KUKA KRL program: f1_Kuka_APT231T02S31.SRC

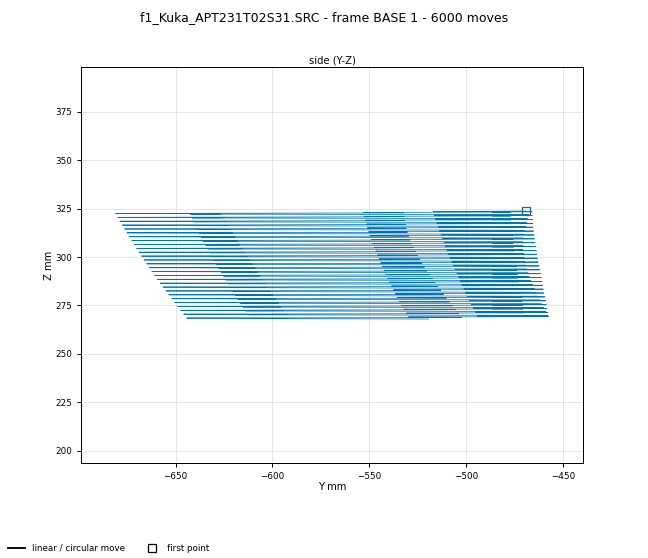
[picture p0: tool path of f1_Kuka_APT231T02S31.SRC in frame BASE 1, 6000 of 6001 moves have a stored position in this frame; points joined in program order, loops and branches not executed]
&ACCESS RVP
&REL 2
&PARAM TEMPLATE = C:\KRC\Roboter\Template\vorgabe
&PARAM EDITMASK = *
DEF f1_Kuka_APT231T02S31()


;FOLD INI;%{PE}%V3.2.0,%MKUKATPBASIS,%CINIT,%VCOMMON,%P
  ;FOLD BAS INI;%{E}%V3.2.0,%MKUKATPBASIS,%CINIT,%VINIT,%P
    GLOBAL INTERRUPT DECL 3 WHEN $STOPMESS==TRUE DO IR_STOPM ( )
    INTERRUPT ON 3
    BAS (#INITMOV,0 )
  ;ENDFOLD (BAS INI)
  ;FOLD USER INI;%{E}%V3.2.0,%MKUKATPUSER,%CINIT,%VINIT,%P
    ;Make your modifications here
  ;ENDFOLD (USER INI)
;ENDFOLD (INI)


;*** Make Null PTP Move
  PTP $pos_act

;*** Auto Load The Correct TOOL Data
  $tool=tool_data[2]

;*** Auto Load The Correct BASE Data
  $base=base_data[1]

  $ADVANCE = 5

;*** Restate Last Velocity
MMPM(30000.0)
SetRPM(8000)
LIN {X 0.027,Y -469.102,Z 323.706,A 0.000,B 0.000,C 90.000,E1 163.015} C_DIS
LIN {X -0.054,Y -471.891,Z 323.687,A 0.000,B 0.000,C 90.000,E1 159.571} C_DIS
LIN {X 0.052,Y -475.505,Z 323.669,A 0.000,B 0.000,C 90.000,E1 156.433} C_DIS
LIN {X 0.015,Y -479.747,Z 323.654,A 0.000,B 0.000,C 90.000,E1 153.640} C_DIS
LIN {X -0.289,Y -483.697,Z 323.642,A 0.000,B 0.000,C 90.000,E1 151.513} C_DIS
LIN {X -0.138,Y -490.881,Z 323.623,A 0.000,B 0.000,C 90.000,E1 148.122} C_DIS
LIN {X -0.106,Y -495.482,Z 323.613,A 0.000,B 0.000,C 90.000,E1 146.294} C_DIS
LIN {X -0.238,Y -500.846,Z 323.601,A 0.000,B 0.000,C 90.000,E1 144.196} C_DIS
LIN {X -0.122,Y -504.629,Z 323.593,A 0.000,B 0.000,C 90.000,E1 142.683} C_DIS
LIN {X 0.166,Y -507.447,Z 323.586,A 0.000,B 0.000,C 90.000,E1 141.457} C_DIS
LIN {X -0.132,Y -509.344,Z 323.581,A 0.000,B 0.000,C 90.000,E1 140.598} C_DIS
LIN {X 0.150,Y -511.693,Z 323.574,A 0.000,B 0.000,C 90.000,E1 139.380} C_DIS
LIN {X -0.165,Y -513.302,Z 323.570,A 0.000,B 0.000,C 90.000,E1 138.528} C_DIS
LIN {X 0.005,Y -514.265,Z 323.566,A 0.000,B 0.000,C 90.000,E1 137.919} C_DIS
LIN {X 0.095,Y -515.410,Z 323.561,A 0.000,B 0.000,C 90.000,E1 137.025} C_DIS
LIN {X 0.170,Y -516.215,Z 323.556,A 0.000,B 0.000,C 90.000,E1 136.134} C_DIS
LIN {X -0.015,Y -516.616,Z 323.553,A 0.000,B 0.000,C 90.000,E1 135.567} C_DIS
LIN {X -0.015,Y -516.959,Z 323.547,A 0.000,B 0.000,C 90.000,E1 134.393} C_DIS
LIN {X 0.093,Y -516.892,Z 323.542,A 0.000,B 0.000,C 90.000,E1 133.500} C_DIS
LIN {X 0.111,Y -516.371,Z 323.535,A 0.000,B 0.000,C 90.000,E1 132.324} C_DIS
LIN {X -0.152,Y -515.651,Z 323.530,A 0.000,B 0.000,C 90.000,E1 131.472} C_DIS
LIN {X -0.166,Y -514.311,Z 323.524,A 0.000,B 0.000,C 90.000,E1 130.297} C_DIS
LIN {X -0.225,Y -512.354,Z 323.516,A 0.000,B 0.000,C 90.000,E1 128.830} C_DIS
LIN {X 0.087,Y -510.241,Z 323.507,A 0.000,B 0.000,C 90.000,E1 127.317} C_DIS
LIN {X 0.041,Y -508.579,Z 323.501,A 0.000,B 0.000,C 90.000,E1 126.137} C_DIS
LIN {X 0.169,Y -507.164,Z 323.496,A 0.000,B 0.000,C 90.000,E1 125.231} C_DIS
LIN {X -0.211,Y -504.512,Z 323.488,A 0.000,B 0.000,C 90.000,E1 123.785} C_DIS
LIN {X 0.180,Y -502.175,Z 323.481,A 0.000,B 0.000,C 90.000,E1 122.546} C_DIS
LIN {X 0.128,Y -499.142,Z 323.473,A 0.000,B 0.000,C 90.000,E1 121.052} C_DIS
LIN {X 0.190,Y -496.035,Z 323.464,A 0.000,B 0.000,C 90.000,E1 119.539} C_DIS
LIN {X 0.194,Y -492.872,Z 323.456,A 0.000,B 0.000,C 90.000,E1 118.025} C_DIS
LIN {X -0.096,Y -489.685,Z 323.447,A 0.000,B 0.000,C 90.000,E1 116.539} C_DIS
LIN {X -0.219,Y -486.506,Z 323.439,A 0.000,B 0.000,C 90.000,E1 115.027} C_DIS
LIN {X 0.048,Y -483.203,Z 323.430,A 0.000,B 0.000,C 90.000,E1 113.462} C_DIS
LIN {X 0.246,Y -479.874,Z 323.422,A 0.000,B 0.000,C 90.000,E1 111.897} C_DIS
LIN {X 0.024,Y -476.568,Z 323.413,A 0.000,B 0.000,C 90.000,E1 110.375} C_DIS
LIN {X -0.039,Y -474.512,Z 323.408,A 0.000,B 0.000,C 90.000,E1 109.450} C_DIS
LIN {X -0.150,Y -469.589,Z 323.396,A 0.000,B 0.000,C 90.000,E1 107.275} C_DIS
LIN {X -0.199,Y -466.672,Z 323.389,A 0.000,B 0.000,C 90.000,E1 106.024} C_DIS
LIN {X 0.061,Y -465.888,Z 323.387,A 0.000,B 0.000,C 90.000,E1 105.662} C_DIS
LIN {X 0.021,Y -465.881,Z 323.387,A 0.000,B 0.000,C 90.000,E1 105.662} C_DIS
LIN {X -0.090,Y -467.389,Z 323.384,A 0.000,B 0.000,C 90.000,E1 105.064} C_DIS
LIN {X 0.166,Y -468.029,Z 323.382,A 0.000,B 0.000,C 90.000,E1 104.717} C_DIS
LIN {X 0.143,Y -476.239,Z 323.356,A 0.000,B 0.000,C 90.000,E1 100.018} C_DIS
LIN {X -0.072,Y -482.133,Z 323.330,A 0.000,B 0.000,C 90.000,E1 95.391} C_DIS
LIN {X 0.164,Y -485.530,Z 323.304,A 0.000,B 0.000,C 90.000,E1 90.745} C_DIS
LIN {X 0.196,Y -486.380,Z 323.280,A 0.000,B 0.000,C 90.000,E1 86.445} C_DIS
LIN {X 0.020,Y -486.349,Z 323.279,A 0.000,B 0.000,C 90.000,E1 86.159} C_DIS
LIN {X 0.099,Y -484.663,Z 323.253,A 0.000,B 0.000,C 90.000,E1 81.546} C_DIS
LIN {X -0.011,Y -480.582,Z 323.227,A 0.000,B 0.000,C 90.000,E1 76.937} C_DIS
LIN {X 0.168,Y -479.655,Z 323.224,A 0.000,B 0.000,C 90.000,E1 76.297} C_DIS
LIN {X 0.002,Y -477.055,Z 323.214,A 0.000,B 0.000,C 90.000,E1 74.574} C_DIS
LIN {X -0.038,Y -477.056,Z 323.214,A 0.000,B 0.000,C 90.000,E1 74.574} C_DIS
LIN {X -0.110,Y -479.157,Z 323.210,A 0.000,B 0.000,C 90.000,E1 73.850} C_DIS
LIN {X 0.001,Y -482.530,Z 323.203,A 0.000,B 0.000,C 90.000,E1 72.598} C_DIS
LIN {X 0.163,Y -486.664,Z 323.195,A 0.000,B 0.000,C 90.000,E1 71.040} C_DIS
LIN {X 0.125,Y -491.697,Z 323.185,A 0.000,B 0.000,C 90.000,E1 69.209} C_DIS
LIN {X -0.023,Y -497.656,Z 323.173,A 0.000,B 0.000,C 90.000,E1 67.102} C_DIS
LIN {X -0.170,Y -501.972,Z 323.164,A 0.000,B 0.000,C 90.000,E1 65.613} C_DIS
LIN {X -0.102,Y -507.999,Z 323.153,A 0.000,B 0.000,C 90.000,E1 63.512} C_DIS
LIN {X -0.093,Y -514.007,Z 323.141,A 0.000,B 0.000,C 90.000,E1 61.435} C_DIS
LIN {X 0.030,Y -518.258,Z 323.133,A 0.000,B 0.000,C 90.000,E1 59.950} C_DIS
LIN {X -0.026,Y -523.352,Z 323.123,A 0.000,B 0.000,C 90.000,E1 58.201} C_DIS
LIN {X 0.318,Y -528.367,Z 323.114,A 0.000,B 0.000,C 90.000,E1 56.421} C_DIS
LIN {X -0.074,Y -531.598,Z 323.107,A 0.000,B 0.000,C 90.000,E1 55.308} C_DIS
LIN {X 0.006,Y -535.465,Z 323.099,A 0.000,B 0.000,C 90.000,E1 53.863} C_DIS
LIN {X 0.012,Y -537.610,Z 323.095,A 0.000,B 0.000,C 90.000,E1 53.004} C_DIS
LIN {X 0.054,Y -540.270,Z 323.088,A 0.000,B 0.000,C 90.000,E1 51.859} C_DIS
LIN {X 0.024,Y -542.118,Z 323.083,A 0.000,B 0.000,C 90.000,E1 51.009} C_DIS
LIN {X -0.292,Y -544.439,Z 323.077,A 0.000,B 0.000,C 90.000,E1 49.908} C_DIS
LIN {X -0.227,Y -546.470,Z 323.071,A 0.000,B 0.000,C 90.000,E1 48.771} C_DIS
LIN {X -0.170,Y -547.848,Z 323.066,A 0.000,B 0.000,C 90.000,E1 47.919} C_DIS
LIN {X -0.062,Y -549.476,Z 323.060,A 0.000,B 0.000,C 90.000,E1 46.782} C_DIS
LIN {X -0.375,Y -550.552,Z 323.055,A 0.000,B 0.000,C 90.000,E1 45.972} C_DIS
LIN {X 0.106,Y -551.383,Z 323.051,A 0.000,B 0.000,C 90.000,E1 45.081} C_DIS
LIN {X 0.242,Y -552.179,Z 323.044,A 0.000,B 0.000,C 90.000,E1 43.947} C_DIS
LIN {X -0.043,Y -552.619,Z 323.040,A 0.000,B 0.000,C 90.000,E1 43.137} C_DIS
LIN {X -0.224,Y -553.008,Z 323.032,A 0.000,B 0.000,C 90.000,E1 41.757} C_DIS
LIN {X -0.038,Y -552.919,Z 323.026,A 0.000,B 0.000,C 90.000,E1 40.620} C_DIS
LIN {X 0.081,Y -552.620,Z 323.021,A 0.000,B 0.000,C 90.000,E1 39.769} C_DIS
LIN {X -0.098,Y -551.998,Z 323.015,A 0.000,B 0.000,C 90.000,E1 38.669} C_DIS
LIN {X -0.168,Y -550.648,Z 323.005,A 0.000,B 0.000,C 90.000,E1 36.996} C_DIS
LIN {X -0.208,Y -549.234,Z 322.998,A 0.000,B 0.000,C 90.000,E1 35.598} C_DIS
LIN {X -0.221,Y -547.381,Z 322.988,A 0.000,B 0.000,C 90.000,E1 33.913} C_DIS
LIN {X -0.095,Y -545.408,Z 322.977,A 0.000,B 0.000,C 90.000,E1 31.926} C_DIS
LIN {X 0.137,Y -543.757,Z 322.968,A 0.000,B 0.000,C 90.000,E1 30.207} C_DIS
LIN {X -0.139,Y -542.253,Z 322.958,A 0.000,B 0.000,C 90.000,E1 28.537} C_DIS
LIN {X -0.029,Y -540.418,Z 322.947,A 0.000,B 0.000,C 90.000,E1 26.539} C_DIS
LIN {X 0.105,Y -539.127,Z 322.940,A 0.000,B 0.000,C 90.000,E1 25.103} C_DIS
LIN {X -0.102,Y -537.376,Z 322.928,A 0.000,B 0.000,C 90.000,E1 23.131} C_DIS
LIN {X 0.202,Y -535.858,Z 322.917,A 0.000,B 0.000,C 90.000,E1 21.099} C_DIS
LIN {X -0.219,Y -534.704,Z 322.906,A 0.000,B 0.000,C 90.000,E1 19.141} C_DIS
LIN {X -0.030,Y -533.865,Z 322.897,A 0.000,B 0.000,C 90.000,E1 17.402} C_DIS
LIN {X 0.184,Y -533.065,Z 322.886,A 0.000,B 0.000,C 90.000,E1 15.371} C_DIS
LIN {X -0.243,Y -532.386,Z 322.873,A 0.000,B 0.000,C 90.000,E1 13.119} C_DIS
LIN {X -0.020,Y -532.204,Z 322.865,A 0.000,B 0.000,C 90.000,E1 11.658} C_DIS
LIN {X -0.192,Y -532.327,Z 322.852,A 0.000,B 0.000,C 90.000,E1 9.378} C_DIS
LIN {X -0.064,Y -532.681,Z 322.841,A 0.000,B 0.000,C 90.000,E1 7.352} C_DIS
LIN {X -0.025,Y -533.291,Z 322.831,A 0.000,B 0.000,C 90.000,E1 5.625} C_DIS
LIN {X 0.031,Y -534.797,Z 322.815,A 0.000,B 0.000,C 90.000,E1 2.751} C_DIS
LIN {X 0.050,Y -536.091,Z 322.804,A 0.000,B 0.000,C 90.000,E1 0.745} C_DIS
LIN {X -0.247,Y -538.748,Z 322.786,A 0.000,B 0.000,C 90.000,E1 357.535} C_DIS
LIN {X -0.172,Y -540.033,Z 322.780,A 0.000,B 0.000,C 90.000,E1 356.388} C_DIS
LIN {X -0.025,Y -541.507,Z 322.772,A 0.000,B 0.000,C 90.000,E1 354.951} C_DIS
LIN {X 0.218,Y -543.517,Z 322.763,A 0.000,B 0.000,C 90.000,E1 353.223} C_DIS
LIN {X -0.103,Y -549.183,Z 322.745,A 0.000,B 0.000,C 90.000,E1 350.151} C_DIS
LIN {X 0.036,Y -553.333,Z 322.734,A 0.000,B 0.000,C 90.000,E1 348.173} C_DIS
LIN {X 0.116,Y -556.849,Z 322.727,A 0.000,B 0.000,C 90.000,E1 346.769} C_DIS
LIN {X -0.030,Y -558.482,Z 322.724,A 0.000,B 0.000,C 90.000,E1 346.228} C_DIS
LIN {X -0.204,Y -564.703,Z 322.711,A 0.000,B 0.000,C 90.000,E1 344.031} C_DIS
LIN {X 0.153,Y -570.395,Z 322.701,A 0.000,B 0.000,C 90.000,E1 342.072} C_DIS
LIN {X -0.088,Y -574.524,Z 322.693,A 0.000,B 0.000,C 90.000,E1 340.732} C_DIS
LIN {X 0.131,Y -579.485,Z 322.684,A 0.000,B 0.000,C 90.000,E1 339.082} C_DIS
LIN {X 0.063,Y -587.372,Z 322.670,A 0.000,B 0.000,C 90.000,E1 336.666} C_DIS
LIN {X 0.026,Y -594.654,Z 322.659,A 0.000,B 0.000,C 90.000,E1 334.537} C_DIS
LIN {X 0.043,Y -600.333,Z 322.650,A 0.000,B 0.000,C 90.000,E1 332.948} C_DIS
LIN {X -0.025,Y -604.988,Z 322.642,A 0.000,B 0.000,C 90.000,E1 331.641} C_DIS
LIN {X 0.161,Y -612.519,Z 322.631,A 0.000,B 0.000,C 90.000,E1 329.537} C_DIS
LIN {X 0.091,Y -617.314,Z 322.624,A 0.000,B 0.000,C 90.000,E1 328.250} C_DIS
LIN {X -0.208,Y -620.931,Z 322.618,A 0.000,B 0.000,C 90.000,E1 327.248} C_DIS
LIN {X 0.411,Y -623.525,Z 322.614,A 0.000,B 0.000,C 90.000,E1 326.421} C_DIS
LIN {X 0.002,Y -627.602,Z 322.607,A 0.000,B 0.000,C 90.000,E1 325.182} C_DIS
LIN {X 0.016,Y -631.423,Z 322.600,A 0.000,B 0.000,C 90.000,E1 323.909} C_DIS
LIN {X 0.092,Y -635.010,Z 322.593,A 0.000,B 0.000,C 90.000,E1 322.637} C_DIS
LIN {X 0.111,Y -638.547,Z 322.586,A 0.000,B 0.000,C 90.000,E1 321.376} C_DIS
LIN {X 0.013,Y -644.305,Z 322.574,A 0.000,B 0.000,C 90.000,E1 319.380} C_DIS
LIN {X -0.300,Y -647.920,Z 322.567,A 0.000,B 0.000,C 90.000,E1 318.162} C_DIS
LIN {X 0.166,Y -654.639,Z 322.555,A 0.000,B 0.000,C 90.000,E1 315.891} C_DIS
LIN {X 0.020,Y -657.734,Z 322.550,A 0.000,B 0.000,C 90.000,E1 314.919} C_DIS
LIN {X -0.128,Y -662.085,Z 322.541,A 0.000,B 0.000,C 90.000,E1 313.461} C_DIS
LIN {X -0.160,Y -665.485,Z 322.535,A 0.000,B 0.000,C 90.000,E1 312.243} C_DIS
LIN {X 0.316,Y -668.009,Z 322.529,A 0.000,B 0.000,C 90.000,E1 311.229} C_DIS
LIN {X -0.128,Y -670.426,Z 322.524,A 0.000,B 0.000,C 90.000,E1 310.297} C_DIS
LIN {X 0.069,Y -673.743,Z 322.516,A 0.000,B 0.000,C 90.000,E1 308.830} C_DIS
LIN {X -0.209,Y -676.138,Z 322.509,A 0.000,B 0.000,C 90.000,E1 307.649} C_DIS
LIN {X -0.067,Y -677.435,Z 322.505,A 0.000,B 0.000,C 90.000,E1 306.916} C_DIS
LIN {X 0.229,Y -678.546,Z 322.501,A 0.000,B 0.000,C 90.000,E1 306.171} C_DIS
LIN {X -0.162,Y -679.263,Z 322.498,A 0.000,B 0.000,C 90.000,E1 305.724} C_DIS
LIN {X 0.164,Y -680.186,Z 322.493,A 0.000,B 0.000,C 90.000,E1 304.739} C_DIS
LIN {X -0.058,Y -680.684,Z 322.489,A 0.000,B 0.000,C 90.000,E1 304.040} C_DIS
LIN {X -0.098,Y -680.975,Z 322.484,A 0.000,B 0.000,C 90.000,E1 303.086} C_DIS
LIN {X 0.256,Y -680.873,Z 322.480,A 0.000,B 0.000,C 90.000,E1 302.339} C_DIS
LIN {X 0.218,Y -680.259,Z 322.475,A 0.000,B 0.000,C 90.000,E1 301.386} C_DIS
LIN {X 0.211,Y -679.554,Z 322.471,A 0.000,B 0.000,C 90.000,E1 300.669} C_DIS
LIN {X -0.384,Y -678.523,Z 322.467,A 0.000,B 0.000,C 90.000,E1 300.001} C_DIS
LIN {X -0.067,Y -677.277,Z 322.463,A 0.000,B 0.000,C 90.000,E1 299.255} C_DIS
LIN {X 0.085,Y -675.286,Z 322.457,A 0.000,B 0.000,C 90.000,E1 298.281} C_DIS
LIN {X 0.082,Y -672.489,Z 322.451,A 0.000,B 0.000,C 90.000,E1 297.078} C_DIS
LIN {X 0.177,Y -670.114,Z 322.445,A 0.000,B 0.000,C 90.000,E1 296.104} C_DIS
LIN {X -0.323,Y -664.969,Z 322.434,A 0.000,B 0.000,C 90.000,E1 294.207} C_DIS
LIN {X 0.120,Y -661.586,Z 322.428,A 0.000,B 0.000,C 90.000,E1 292.950} C_DIS
LIN {X 0.246,Y -658.195,Z 322.421,A 0.000,B 0.000,C 90.000,E1 291.716} C_DIS
LIN {X 0.278,Y -653.533,Z 322.411,A 0.000,B 0.000,C 90.000,E1 289.993} C_DIS
LIN {X -0.231,Y -649.159,Z 322.402,A 0.000,B 0.000,C 90.000,E1 288.308} C_DIS
LIN {X -0.059,Y -645.642,Z 322.393,A 0.000,B 0.000,C 90.000,E1 286.804} C_DIS
LIN {X -0.126,Y -641.800,Z 322.384,A 0.000,B 0.000,C 90.000,E1 285.064} C_DIS
LIN {X -0.162,Y -637.875,Z 322.373,A 0.000,B 0.000,C 90.000,E1 283.063} C_DIS
LIN {X 0.279,Y -633.512,Z 322.357,A 0.000,B 0.000,C 90.000,E1 280.254} C_DIS
LIN {X -0.172,Y -629.759,Z 322.339,A 0.000,B 0.000,C 90.000,E1 277.004} C_DIS
LIN {X -0.269,Y -627.978,Z 322.325,A 0.000,B 0.000,C 90.000,E1 274.473} C_DIS
LIN {X 0.138,Y -627.011,Z 322.311,A 0.000,B 0.000,C 90.000,E1 271.892} C_DIS
LIN {X 0.153,Y -626.803,Z 322.298,A 0.000,B 0.000,C 90.000,E1 269.599} C_DIS
LIN {X -0.184,Y -627.189,Z 322.287,A 0.000,B 0.000,C 90.000,E1 267.593} C_DIS
LIN {X 0.258,Y -628.481,Z 322.272,A 0.000,B 0.000,C 90.000,E1 265.008} C_DIS
LIN {X 0.243,Y -630.368,Z 322.258,A 0.000,B 0.000,C 90.000,E1 262.470} C_DIS
LIN {X 0.233,Y -632.319,Z 322.247,A 0.000,B 0.000,C 90.000,E1 260.443} C_DIS
LIN {X 0.236,Y -633.993,Z 322.239,A 0.000,B 0.000,C 90.000,E1 258.926} C_DIS
LIN {X -0.251,Y -637.011,Z 322.226,A 0.000,B 0.000,C 90.000,E1 256.700} C_DIS
LIN {X 0.139,Y -638.757,Z 322.219,A 0.000,B 0.000,C 90.000,E1 255.408} C_DIS
LIN {X 0.262,Y -639.958,Z 322.213,A 0.000,B 0.000,C 90.000,E1 254.393} C_DIS
LIN {X 0.081,Y -641.307,Z 322.205,A 0.000,B 0.000,C 90.000,E1 252.906} C_DIS
LIN {X -0.376,Y -642.020,Z 322.200,A 0.000,B 0.000,C 90.000,E1 251.945} C_DIS
LIN {X 0.151,Y -642.366,Z 322.195,A 0.000,B 0.000,C 90.000,E1 251.148} C_DIS
LIN {X -0.130,Y -642.448,Z 322.191,A 0.000,B 0.000,C 90.000,E1 250.423} C_DIS
LIN {X 0.188,Y -642.219,Z 322.187,A 0.000,B 0.000,C 90.000,E1 249.645} C_DIS
LIN {X 0.068,Y -641.972,Z 322.184,A 0.000,B 0.000,C 90.000,E1 249.156} C_DIS
LIN {X 0.180,Y -641.650,Z 322.182,A 0.000,B 0.000,C 90.000,E1 248.646} C_DIS
LIN {X -0.124,Y -640.780,Z 322.177,A 0.000,B 0.000,C 90.000,E1 247.922} C_DIS
LIN {X -0.009,Y -640.107,Z 322.175,A 0.000,B 0.000,C 90.000,E1 247.411} C_DIS
LIN {X -0.086,Y -638.795,Z 322.170,A 0.000,B 0.000,C 90.000,E1 246.666} C_DIS
LIN {X -0.178,Y -637.316,Z 322.166,A 0.000,B 0.000,C 90.000,E1 245.921} C_DIS
LIN {X -0.024,Y -635.637,Z 322.162,A 0.000,B 0.000,C 90.000,E1 245.153} C_DIS
LIN {X -0.197,Y -634.439,Z 322.159,A 0.000,B 0.000,C 90.000,E1 244.665} C_DIS
LIN {X -0.070,Y -632.314,Z 322.155,A 0.000,B 0.000,C 90.000,E1 243.896} C_DIS
LIN {X 0.096,Y -628.417,Z 322.148,A 0.000,B 0.000,C 90.000,E1 242.615} C_DIS
LIN {X -0.053,Y -623.547,Z 322.139,A 0.000,B 0.000,C 90.000,E1 241.101} C_DIS
LIN {X 0.257,Y -619.423,Z 322.132,A 0.000,B 0.000,C 90.000,E1 239.793} C_DIS
LIN {X 0.213,Y -613.578,Z 322.122,A 0.000,B 0.000,C 90.000,E1 237.995} C_DIS
LIN {X 0.128,Y -609.344,Z 322.115,A 0.000,B 0.000,C 90.000,E1 236.707} C_DIS
LIN {X 0.039,Y -605.897,Z 322.109,A 0.000,B 0.000,C 90.000,E1 235.674} C_DIS
LIN {X 0.155,Y -601.638,Z 322.102,A 0.000,B 0.000,C 90.000,E1 234.356} C_DIS
LIN {X -0.177,Y -598.101,Z 322.096,A 0.000,B 0.000,C 90.000,E1 233.336} C_DIS
LIN {X -0.074,Y -594.367,Z 322.090,A 0.000,B 0.000,C 90.000,E1 232.271} C_DIS
LIN {X 0.056,Y -586.091,Z 322.077,A 0.000,B 0.000,C 90.000,E1 229.865} C_DIS
LIN {X 0.067,Y -578.938,Z 322.065,A 0.000,B 0.000,C 90.000,E1 227.715} C_DIS
LIN {X -0.089,Y -574.613,Z 322.058,A 0.000,B 0.000,C 90.000,E1 226.377} C_DIS
LIN {X -0.024,Y -571.037,Z 322.052,A 0.000,B 0.000,C 90.000,E1 225.283} C_DIS
LIN {X -0.042,Y -564.046,Z 322.039,A 0.000,B 0.000,C 90.000,E1 223.095} C_DIS
LIN {X 0.011,Y -558.842,Z 322.030,A 0.000,B 0.000,C 90.000,E1 221.434} C_DIS
LIN {X 0.343,Y -554.568,Z 322.023,A 0.000,B 0.000,C 90.000,E1 220.011} C_DIS
LIN {X -0.065,Y -548.553,Z 322.012,A 0.000,B 0.000,C 90.000,E1 218.096} C_DIS
LIN {X 0.173,Y -544.358,Z 322.004,A 0.000,B 0.000,C 90.000,E1 216.664} C_DIS
LIN {X 0.095,Y -536.316,Z 321.988,A 0.000,B 0.000,C 90.000,E1 213.833} C_DIS
LIN {X -0.086,Y -531.057,Z 321.977,A 0.000,B 0.000,C 90.000,E1 211.848} C_DIS
LIN {X 0.226,Y -526.102,Z 321.966,A 0.000,B 0.000,C 90.000,E1 209.795} C_DIS
LIN {X 0.157,Y -521.181,Z 321.954,A 0.000,B 0.000,C 90.000,E1 207.769} C_DIS
LIN {X 0.185,Y -516.436,Z 321.943,A 0.000,B 0.000,C 90.000,E1 205.720} C_DIS
LIN {X 0.219,Y -512.550,Z 321.933,A 0.000,B 0.000,C 90.000,E1 203.951} C_DIS
LIN {X -0.149,Y -509.241,Z 321.925,A 0.000,B 0.000,C 90.000,E1 202.514} C_DIS
LIN {X -0.198,Y -505.271,Z 321.915,A 0.000,B 0.000,C 90.000,E1 200.737} C_DIS
LIN {X 0.064,Y -502.096,Z 321.907,A 0.000,B 0.000,C 90.000,E1 199.214} C_DIS
LIN {X 0.166,Y -498.345,Z 321.897,A 0.000,B 0.000,C 90.000,E1 197.402} C_DIS
LIN {X -0.031,Y -493.606,Z 321.883,A 0.000,B 0.000,C 90.000,E1 195.009} C_DIS
LIN {X -0.147,Y -489.370,Z 321.870,A 0.000,B 0.000,C 90.000,E1 192.591} C_DIS
LIN {X 0.009,Y -485.745,Z 321.858,A 0.000,B 0.000,C 90.000,E1 190.433} C_DIS
LIN {X 0.062,Y -482.253,Z 321.846,A 0.000,B 0.000,C 90.000,E1 188.276} C_DIS
LIN {X -0.073,Y -478.262,Z 321.831,A 0.000,B 0.000,C 90.000,E1 185.511} C_DIS
LIN {X -0.112,Y -474.343,Z 321.813,A 0.000,B 0.000,C 90.000,E1 182.407} C_DIS
LIN {X 0.173,Y -470.180,Z 321.789,A 0.000,B 0.000,C 90.000,E1 177.993} C_DIS
LIN {X -0.148,Y -468.147,Z 321.768,A 0.000,B 0.000,C 90.000,E1 174.261} C_DIS
LIN {X 0.156,Y -467.503,Z 321.747,A 0.000,B 0.000,C 90.000,E1 170.443} C_DIS
LIN {X -0.152,Y -467.871,Z 321.731,A 0.000,B 0.000,C 90.000,E1 167.645} C_DIS
LIN {X 0.119,Y -469.076,Z 321.714,A 0.000,B 0.000,C 90.000,E1 164.464} C_DIS
LIN {X 0.007,Y -469.941,Z 321.705,A 0.000,B 0.000,C 90.000,E1 162.906} C_DIS
LIN {X 0.144,Y -472.374,Z 321.688,A 0.000,B 0.000,C 90.000,E1 159.752} C_DIS
LIN {X -0.163,Y -475.826,Z 321.670,A 0.000,B 0.000,C 90.000,E1 156.666} C_DIS
LIN {X 0.045,Y -479.902,Z 321.655,A 0.000,B 0.000,C 90.000,E1 153.845} C_DIS
LIN {X -0.047,Y -484.253,Z 321.641,A 0.000,B 0.000,C 90.000,E1 151.385} C_DIS
LIN {X -0.124,Y -490.621,Z 321.624,A 0.000,B 0.000,C 90.000,E1 148.329} C_DIS
LIN {X -0.099,Y -495.085,Z 321.614,A 0.000,B 0.000,C 90.000,E1 146.501} C_DIS
LIN {X -0.243,Y -500.328,Z 321.602,A 0.000,B 0.000,C 90.000,E1 144.402} C_DIS
LIN {X 0.155,Y -504.803,Z 321.592,A 0.000,B 0.000,C 90.000,E1 142.557} C_DIS
LIN {X -0.167,Y -506.898,Z 321.587,A 0.000,B 0.000,C 90.000,E1 141.698} C_DIS
LIN {X -0.153,Y -508.790,Z 321.582,A 0.000,B 0.000,C 90.000,E1 140.803} C_DIS
LIN {X -0.207,Y -511.081,Z 321.576,A 0.000,B 0.000,C 90.000,E1 139.622} C_DIS
LIN {X 0.190,Y -512.652,Z 321.571,A 0.000,B 0.000,C 90.000,E1 138.690} C_DIS
LIN {X 0.013,Y -513.621,Z 321.567,A 0.000,B 0.000,C 90.000,E1 138.119} C_DIS
LIN {X 0.061,Y -514.748,Z 321.562,A 0.000,B 0.000,C 90.000,E1 137.229} C_DIS
LIN {X -0.223,Y -515.579,Z 321.558,A 0.000,B 0.000,C 90.000,E1 136.377} C_DIS
LIN {X -0.143,Y -516.147,Z 321.553,A 0.000,B 0.000,C 90.000,E1 135.486} C_DIS
LIN {X 0.219,Y -516.362,Z 321.546,A 0.000,B 0.000,C 90.000,E1 134.271} C_DIS
LIN {X -0.048,Y -516.259,Z 321.541,A 0.000,B 0.000,C 90.000,E1 133.419} C_DIS
LIN {X -0.040,Y -515.597,Z 321.535,A 0.000,B 0.000,C 90.000,E1 132.243} C_DIS
LIN {X -0.234,Y -515.152,Z 321.531,A 0.000,B 0.000,C 90.000,E1 131.676} C_DIS
LIN {X 0.132,Y -513.847,Z 321.525,A 0.000,B 0.000,C 90.000,E1 130.458} C_DIS
LIN {X 0.066,Y -511.918,Z 321.517,A 0.000,B 0.000,C 90.000,E1 128.991} C_DIS
LIN {X 0.054,Y -510.215,Z 321.510,A 0.000,B 0.000,C 90.000,E1 127.810} C_DIS
LIN {X 0.323,Y -508.123,Z 321.502,A 0.000,B 0.000,C 90.000,E1 126.297} C_DIS
LIN {X -0.063,Y -506.248,Z 321.495,A 0.000,B 0.000,C 90.000,E1 125.152} C_DIS
LIN {X -0.041,Y -503.565,Z 321.487,A 0.000,B 0.000,C 90.000,E1 123.658} C_DIS
LIN {X 0.034,Y -501.809,Z 321.482,A 0.000,B 0.000,C 90.000,E1 122.752} C_DIS
LIN {X -0.021,Y -498.798,Z 321.474,A 0.000,B 0.000,C 90.000,E1 121.258} C_DIS
LIN {X -0.118,Y -495.066,Z 321.464,A 0.000,B 0.000,C 90.000,E1 119.461} C_DIS
LIN {X 0.299,Y -491.932,Z 321.455,A 0.000,B 0.000,C 90.000,E1 117.897} C_DIS
LIN {X -0.009,Y -488.768,Z 321.447,A 0.000,B 0.000,C 90.000,E1 116.411} C_DIS
LIN {X -0.135,Y -484.971,Z 321.437,A 0.000,B 0.000,C 90.000,E1 114.591} C_DIS
LIN {X 0.106,Y -480.365,Z 321.425,A 0.000,B 0.000,C 90.000,E1 112.408} C_DIS
LIN {X 0.056,Y -476.459,Z 321.414,A 0.000,B 0.000,C 90.000,E1 110.556} C_DIS
LIN {X -0.037,Y -473.828,Z 321.407,A 0.000,B 0.000,C 90.000,E1 109.322} C_DIS
LIN {X -0.171,Y -469.076,Z 321.395,A 0.000,B 0.000,C 90.000,E1 107.149} C_DIS
LIN {X 0.206,Y -465.835,Z 321.387,A 0.000,B 0.000,C 90.000,E1 105.662} C_DIS
LIN {X 0.166,Y -465.837,Z 321.387,A 0.000,B 0.000,C 90.000,E1 105.662} C_DIS
LIN {X -0.251,Y -467.716,Z 321.383,A 0.000,B 0.000,C 90.000,E1 104.954} C_DIS
LIN {X 0.173,Y -475.925,Z 321.357,A 0.000,B 0.000,C 90.000,E1 100.197} C_DIS
LIN {X 0.012,Y -476.360,Z 321.355,A 0.000,B 0.000,C 90.000,E1 99.905} C_DIS
LIN {X -0.031,Y -481.883,Z 321.331,A 0.000,B 0.000,C 90.000,E1 95.568} C_DIS
LIN {X -0.184,Y -482.195,Z 321.329,A 0.000,B 0.000,C 90.000,E1 95.277} C_DIS
LIN {X 0.235,Y -485.370,Z 321.305,A 0.000,B 0.000,C 90.000,E1 90.917} C_DIS
LIN {X 0.059,Y -485.531,Z 321.304,A 0.000,B 0.000,C 90.000,E1 90.630} C_DIS
LIN {X -0.218,Y -486.348,Z 321.281,A 0.000,B 0.000,C 90.000,E1 86.674} C_DIS
LIN {X 0.092,Y -486.369,Z 321.280,A 0.000,B 0.000,C 90.000,E1 86.331} C_DIS
LIN {X -0.226,Y -486.059,Z 321.276,A 0.000,B 0.000,C 90.000,E1 85.755} C_DIS
LIN {X 0.116,Y -484.693,Z 321.254,A 0.000,B 0.000,C 90.000,E1 81.724} C_DIS
LIN {X -0.016,Y -484.528,Z 321.252,A 0.000,B 0.000,C 90.000,E1 81.432} C_DIS
LIN {X -0.147,Y -480.466,Z 321.227,A 0.000,B 0.000,C 90.000,E1 76.825} C_DIS
LIN {X -0.161,Y -476.955,Z 321.214,A 0.000,B 0.000,C 90.000,E1 74.519} C_DIS
LIN {X -0.201,Y -476.956,Z 321.214,A 0.000,B 0.000,C 90.000,E1 74.519} C_DIS
LIN {X 0.172,Y -479.802,Z 321.208,A 0.000,B 0.000,C 90.000,E1 73.378} C_DIS
LIN {X 0.133,Y -484.705,Z 321.198,A 0.000,B 0.000,C 90.000,E1 71.529} C_DIS
LIN {X 0.047,Y -489.671,Z 321.187,A 0.000,B 0.000,C 90.000,E1 69.699} C_DIS
LIN {X 0.257,Y -494.731,Z 321.177,A 0.000,B 0.000,C 90.000,E1 67.847} C_DIS
LIN {X 0.064,Y -499.007,Z 321.169,A 0.000,B 0.000,C 90.000,E1 66.357} C_DIS
LIN {X 0.076,Y -502.460,Z 321.162,A 0.000,B 0.000,C 90.000,E1 65.153} C_DIS
LIN {X -0.143,Y -507.649,Z 321.152,A 0.000,B 0.000,C 90.000,E1 63.384} C_DIS
LIN {X -0.145,Y -513.662,Z 321.141,A 0.000,B 0.000,C 90.000,E1 61.307} C_DIS
LIN {X 0.229,Y -517.903,Z 321.132,A 0.000,B 0.000,C 90.000,E1 59.793} C_DIS
LIN {X -0.099,Y -523.042,Z 321.123,A 0.000,B 0.000,C 90.000,E1 58.074} C_DIS
LIN {X 0.234,Y -528.038,Z 321.113,A 0.000,B 0.000,C 90.000,E1 56.294} C_DIS
LIN {X -0.166,Y -531.256,Z 321.107,A 0.000,B 0.000,C 90.000,E1 55.182} C_DIS
LIN {X 0.218,Y -535.119,Z 321.099,A 0.000,B 0.000,C 90.000,E1 53.703} C_DIS
LIN {X 0.231,Y -537.960,Z 321.092,A 0.000,B 0.000,C 90.000,E1 52.557} C_DIS
LIN {X -0.142,Y -540.522,Z 321.086,A 0.000,B 0.000,C 90.000,E1 51.457} C_DIS
LIN {X 0.284,Y -542.944,Z 321.080,A 0.000,B 0.000,C 90.000,E1 50.275} C_DIS
LIN {X -0.026,Y -545.067,Z 321.073,A 0.000,B 0.000,C 90.000,E1 49.175} C_DIS
LIN {X 0.043,Y -547.002,Z 321.067,A 0.000,B 0.000,C 90.000,E1 48.038} C_DIS
LIN {X -0.302,Y -548.260,Z 321.062,A 0.000,B 0.000,C 90.000,E1 47.229} C_DIS
LIN {X 0.185,Y -549.733,Z 321.056,A 0.000,B 0.000,C 90.000,E1 46.053} C_DIS
LIN {X 0.239,Y -550.345,Z 321.053,A 0.000,B 0.000,C 90.000,E1 45.486} C_DIS
LIN {X -0.060,Y -551.086,Z 321.048,A 0.000,B 0.000,C 90.000,E1 44.676} C_DIS
LIN {X -0.353,Y -551.695,Z 321.044,A 0.000,B 0.000,C 90.000,E1 43.866} C_DIS
LIN {X 0.114,Y -552.055,Z 321.040,A 0.000,B 0.000,C 90.000,E1 43.257} C_DIS
LIN {X 0.304,Y -552.549,Z 321.033,A 0.000,B 0.000,C 90.000,E1 41.838} C_DIS
LIN {X 0.065,Y -552.558,Z 321.026,A 0.000,B 0.000,C 90.000,E1 40.744} C_DIS
LIN {X -0.178,Y -552.361,Z 321.022,A 0.000,B 0.000,C 90.000,E1 39.930} C_DIS
LIN {X -0.295,Y -551.639,Z 321.014,A 0.000,B 0.000,C 90.000,E1 38.543} C_DIS
LIN {X 0.014,Y -550.567,Z 321.006,A 0.000,B 0.000,C 90.000,E1 37.111} C_DIS
LIN {X -0.139,Y -549.186,Z 320.998,A 0.000,B 0.000,C 90.000,E1 35.724} C_DIS
LIN {X -0.158,Y -547.379,Z 320.989,A 0.000,B 0.000,C 90.000,E1 34.040} C_DIS
LIN {X -0.036,Y -545.382,Z 320.978,A 0.000,B 0.000,C 90.000,E1 32.054} C_DIS
LIN {X -0.066,Y -543.468,Z 320.967,A 0.000,B 0.000,C 90.000,E1 30.079} C_DIS
LIN {X 0.130,Y -541.985,Z 320.958,A 0.000,B 0.000,C 90.000,E1 28.359} C_DIS
LIN {X 0.242,Y -540.141,Z 320.947,A 0.000,B 0.000,C 90.000,E1 26.360} C_DIS
LIN {X 0.115,Y -538.844,Z 320.939,A 0.000,B 0.000,C 90.000,E1 24.951} C_DIS
LIN {X 0.165,Y -537.101,Z 320.928,A 0.000,B 0.000,C 90.000,E1 22.950} C_DIS
LIN {X -0.244,Y -535.807,Z 320.918,A 0.000,B 0.000,C 90.000,E1 21.280} C_DIS
LIN {X -0.163,Y -534.617,Z 320.907,A 0.000,B 0.000,C 90.000,E1 19.268} C_DIS
LIN {X 0.189,Y -533.757,Z 320.897,A 0.000,B 0.000,C 90.000,E1 17.511} C_DIS
LIN {X -0.085,Y -532.812,Z 320.885,A 0.000,B 0.000,C 90.000,E1 15.245} C_DIS
LIN {X -0.174,Y -532.244,Z 320.874,A 0.000,B 0.000,C 90.000,E1 13.244} C_DIS
LIN {X 0.161,Y -532.042,Z 320.866,A 0.000,B 0.000,C 90.000,E1 11.771} C_DIS
LIN {X -0.069,Y -532.144,Z 320.851,A 0.000,B 0.000,C 90.000,E1 9.208} C_DIS
LIN {X 0.063,Y -532.523,Z 320.840,A 0.000,B 0.000,C 90.000,E1 7.182} C_DIS
LIN {X 0.106,Y -533.145,Z 320.830,A 0.000,B 0.000,C 90.000,E1 5.454} C_DIS
LIN {X 0.162,Y -534.666,Z 320.814,A 0.000,B 0.000,C 90.000,E1 2.579} C_DIS
LIN {X 0.180,Y -535.925,Z 320.803,A 0.000,B 0.000,C 90.000,E1 0.573} C_DIS
LIN {X -0.247,Y -538.693,Z 320.785,A 0.000,B 0.000,C 90.000,E1 357.249} C_DIS
LIN {X -0.175,Y -539.920,Z 320.778,A 0.000,B 0.000,C 90.000,E1 356.102} C_DIS
LIN {X -0.045,Y -541.071,Z 320.772,A 0.000,B 0.000,C 90.000,E1 354.951} C_DIS
LIN {X 0.115,Y -542.646,Z 320.764,A 0.000,B 0.000,C 90.000,E1 353.514} C_DIS
LIN {X -0.155,Y -548.620,Z 320.745,A 0.000,B 0.000,C 90.000,E1 350.151} C_DIS
LIN {X -0.032,Y -552.739,Z 320.734,A 0.000,B 0.000,C 90.000,E1 348.173} C_DIS
LIN {X 0.159,Y -559.319,Z 320.720,A 0.000,B 0.000,C 90.000,E1 345.644} C_DIS
LIN {X -0.156,Y -564.784,Z 320.710,A 0.000,B 0.000,C 90.000,E1 343.740} C_DIS
LIN {X -0.172,Y -570.450,Z 320.699,A 0.000,B 0.000,C 90.000,E1 341.819} C_DIS
LIN {X 0.135,Y -574.585,Z 320.691,A 0.000,B 0.000,C 90.000,E1 340.423} C_DIS
LIN {X -0.181,Y -579.514,Z 320.682,A 0.000,B 0.000,C 90.000,E1 338.827} C_DIS
LIN {X -0.120,Y -586.582,Z 320.670,A 0.000,B 0.000,C 90.000,E1 336.666} C_DIS
LIN {X -0.181,Y -593.874,Z 320.658,A 0.000,B 0.000,C 90.000,E1 334.537} C_DIS
LIN {X 0.091,Y -599.561,Z 320.650,A 0.000,B 0.000,C 90.000,E1 332.922} C_DIS
LIN {X -0.264,Y -604.225,Z 320.642,A 0.000,B 0.000,C 90.000,E1 331.641} C_DIS
LIN {X -0.058,Y -610.809,Z 320.632,A 0.000,B 0.000,C 90.000,E1 329.793} C_DIS
LIN {X -0.189,Y -616.478,Z 320.624,A 0.000,B 0.000,C 90.000,E1 328.250} C_DIS
LIN {X 0.022,Y -620.140,Z 320.618,A 0.000,B 0.000,C 90.000,E1 327.199} C_DIS
LIN {X 0.087,Y -623.526,Z 320.612,A 0.000,B 0.000,C 90.000,E1 326.167} C_DIS
LIN {X 0.216,Y -626.085,Z 320.608,A 0.000,B 0.000,C 90.000,E1 325.388} C_DIS
LIN {X -0.316,Y -630.732,Z 320.599,A 0.000,B 0.000,C 90.000,E1 323.909} C_DIS
LIN {X -0.254,Y -634.387,Z 320.592,A 0.000,B 0.000,C 90.000,E1 322.637} C_DIS
LIN {X -0.367,Y -639.314,Z 320.583,A 0.000,B 0.000,C 90.000,E1 320.884} C_DIS
LIN {X -0.364,Y -643.681,Z 320.574,A 0.000,B 0.000,C 90.000,E1 319.380} C_DIS
LIN {X 0.224,Y -647.279,Z 320.567,A 0.000,B 0.000,C 90.000,E1 318.081} C_DIS
LIN {X -0.201,Y -653.220,Z 320.556,A 0.000,B 0.000,C 90.000,E1 316.134} C_DIS
LIN {X 0.097,Y -656.339,Z 320.551,A 0.000,B 0.000,C 90.000,E1 315.121} C_DIS
LIN {X -0.067,Y -660.689,Z 320.543,A 0.000,B 0.000,C 90.000,E1 313.662} C_DIS
LIN {X -0.138,Y -663.444,Z 320.537,A 0.000,B 0.000,C 90.000,E1 312.690} C_DIS
LIN {X 0.307,Y -666.030,Z 320.532,A 0.000,B 0.000,C 90.000,E1 311.676} C_DIS
LIN {X -0.092,Y -669.650,Z 320.524,A 0.000,B 0.000,C 90.000,E1 310.253} C_DIS
LIN {X -0.425,Y -672.901,Z 320.516,A 0.000,B 0.000,C 90.000,E1 308.830} C_DIS
LIN {X -0.184,Y -675.298,Z 320.509,A 0.000,B 0.000,C 90.000,E1 307.604} C_DIS
LIN {X -0.043,Y -676.933,Z 320.504,A 0.000,B 0.000,C 90.000,E1 306.629} C_DIS
LIN {X -0.145,Y -678.265,Z 320.498,A 0.000,B 0.000,C 90.000,E1 305.678} C_DIS
LIN {X 0.009,Y -678.983,Z 320.494,A 0.000,B 0.000,C 90.000,E1 304.945} C_DIS
LIN {X 0.338,Y -679.511,Z 320.490,A 0.000,B 0.000,C 90.000,E1 304.199} C_DIS
LIN {X -0.442,Y -679.765,Z 320.488,A 0.000,B 0.000,C 90.000,E1 303.785} C_DIS
LIN {X -0.119,Y -679.833,Z 320.482,A 0.000,B 0.000,C 90.000,E1 302.801} C_DIS
LIN {X -0.142,Y -679.598,Z 320.478,A 0.000,B 0.000,C 90.000,E1 302.084} C_DIS
LIN {X -0.192,Y -678.853,Z 320.473,A 0.000,B 0.000,C 90.000,E1 301.131} C_DIS
LIN {X 0.135,Y -677.973,Z 320.469,A 0.000,B 0.000,C 90.000,E1 300.384} C_DIS
LIN {X 0.110,Y -676.811,Z 320.465,A 0.000,B 0.000,C 90.000,E1 299.667} C_DIS
LIN {X 0.078,Y -675.467,Z 320.461,A 0.000,B 0.000,C 90.000,E1 298.949} C_DIS
LIN {X 0.214,Y -673.338,Z 320.456,A 0.000,B 0.000,C 90.000,E1 297.975} C_DIS
LIN {X -0.106,Y -670.489,Z 320.449,A 0.000,B 0.000,C 90.000,E1 296.796} C_DIS
LIN {X 0.096,Y -668.644,Z 320.445,A 0.000,B 0.000,C 90.000,E1 296.052} C_DIS
LIN {X 0.155,Y -664.760,Z 320.437,A 0.000,B 0.000,C 90.000,E1 294.591} C_DIS
LIN {X -0.146,Y -662.178,Z 320.431,A 0.000,B 0.000,C 90.000,E1 293.643} C_DIS
LIN {X 0.116,Y -658.082,Z 320.423,A 0.000,B 0.000,C 90.000,E1 292.153} C_DIS
LIN {X 0.245,Y -652.737,Z 320.412,A 0.000,B 0.000,C 90.000,E1 290.174} C_DIS
LIN {X -0.079,Y -648.325,Z 320.403,A 0.000,B 0.000,C 90.000,E1 288.471} C_DIS
LIN {X -0.090,Y -644.201,Z 320.393,A 0.000,B 0.000,C 90.000,E1 286.732} C_DIS
LIN {X -0.069,Y -639.391,Z 320.380,A 0.000,B 0.000,C 90.000,E1 284.481} C_DIS
LIN {X 0.018,Y -633.238,Z 320.361,A 0.000,B 0.000,C 90.000,E1 280.950} C_DIS
LIN {X 0.058,Y -629.724,Z 320.345,A 0.000,B 0.000,C 90.000,E1 278.163} C_DIS
LIN {X 0.239,Y -626.844,Z 320.326,A 0.000,B 0.000,C 90.000,E1 274.588} C_DIS
LIN {X -0.140,Y -626.105,Z 320.317,A 0.000,B 0.000,C 90.000,E1 273.094} C_DIS
LIN {X -0.285,Y -625.756,Z 320.310,A 0.000,B 0.000,C 90.000,E1 271.833} C_DIS
LIN {X -0.047,Y -625.602,Z 320.299,A 0.000,B 0.000,C 90.000,E1 269.771} C_DIS
LIN {X -0.072,Y -626.001,Z 320.286,A 0.000,B 0.000,C 90.000,E1 267.478} C_DIS
LIN {X 0.225,Y -627.030,Z 320.275,A 0.000,B 0.000,C 90.000,E1 265.412} C_DIS
LIN {X -0.257,Y -628.608,Z 320.262,A 0.000,B 0.000,C 90.000,E1 263.166} C_DIS
LIN {X -0.118,Y -630.240,Z 320.252,A 0.000,B 0.000,C 90.000,E1 261.376} C_DIS
LIN {X -0.042,Y -632.479,Z 320.241,A 0.000,B 0.000,C 90.000,E1 259.342} C_DIS
LIN {X -0.324,Y -636.144,Z 320.225,A 0.000,B 0.000,C 90.000,E1 256.589} C_DIS
LIN {X 0.205,Y -637.886,Z 320.218,A 0.000,B 0.000,C 90.000,E1 255.283} C_DIS
LIN {X 0.148,Y -639.085,Z 320.213,A 0.000,B 0.000,C 90.000,E1 254.283} C_DIS
LIN {X 0.130,Y -640.439,Z 320.204,A 0.000,B 0.000,C 90.000,E1 252.779} C_DIS
LIN {X 0.274,Y -641.163,Z 320.199,A 0.000,B 0.000,C 90.000,E1 251.764} C_DIS
LIN {X -0.022,Y -641.548,Z 320.195,A 0.000,B 0.000,C 90.000,E1 251.040} C_DIS
LIN {X -0.100,Y -641.602,Z 320.191,A 0.000,B 0.000,C 90.000,E1 250.296} C_DIS
LIN {X 0.262,Y -641.340,Z 320.185,A 0.000,B 0.000,C 90.000,E1 249.263} C_DIS
LIN {X -0.040,Y -640.871,Z 320.181,A 0.000,B 0.000,C 90.000,E1 248.539} C_DIS
LIN {X -0.114,Y -640.071,Z 320.177,A 0.000,B 0.000,C 90.000,E1 247.794} C_DIS
LIN {X -0.002,Y -639.410,Z 320.174,A 0.000,B 0.000,C 90.000,E1 247.283} C_DIS
LIN {X -0.288,Y -637.674,Z 320.168,A 0.000,B 0.000,C 90.000,E1 246.305} C_DIS
LIN {X -0.184,Y -636.672,Z 320.165,A 0.000,B 0.000,C 90.000,E1 245.793} C_DIS
LIN {X -0.034,Y -634.970,Z 320.161,A 0.000,B 0.000,C 90.000,E1 245.025} C_DIS
LIN {X -0.213,Y -633.715,Z 320.158,A 0.000,B 0.000,C 90.000,E1 244.537} C_DIS
LIN {X -0.092,Y -631.569,Z 320.154,A 0.000,B 0.000,C 90.000,E1 243.768} C_DIS
LIN {X 0.060,Y -627.717,Z 320.147,A 0.000,B 0.000,C 90.000,E1 242.487} C_DIS
LIN {X -0.097,Y -622.053,Z 320.137,A 0.000,B 0.000,C 90.000,E1 240.717} C_DIS
LIN {X 0.181,Y -617.937,Z 320.130,A 0.000,B 0.000,C 90.000,E1 239.410} C_DIS
LIN {X 0.132,Y -612.975,Z 320.122,A 0.000,B 0.000,C 90.000,E1 237.867} C_DIS
LIN {X 0.035,Y -608.811,Z 320.114,A 0.000,B 0.000,C 90.000,E1 236.580} C_DIS
LIN {X -0.063,Y -605.406,Z 320.109,A 0.000,B 0.000,C 90.000,E1 235.548} C_DIS
LIN {X -0.098,Y -601.180,Z 320.101,A 0.000,B 0.000,C 90.000,E1 234.242} C_DIS
LIN {X -0.301,Y -597.681,Z 320.095,A 0.000,B 0.000,C 90.000,E1 233.210} C_DIS
LIN {X -0.232,Y -592.085,Z 320.087,A 0.000,B 0.000,C 90.000,E1 231.618} C_DIS
LIN {X -0.169,Y -585.719,Z 320.076,A 0.000,B 0.000,C 90.000,E1 229.747} C_DIS
LIN {X 0.126,Y -579.534,Z 320.066,A 0.000,B 0.000,C 90.000,E1 227.838} C_DIS
LIN {X -0.011,Y -575.268,Z 320.058,A 0.000,B 0.000,C 90.000,E1 226.500} C_DIS
LIN {X 0.069,Y -571.704,Z 320.052,A 0.000,B 0.000,C 90.000,E1 225.405} C_DIS
LIN {X 0.059,Y -564.779,Z 320.040,A 0.000,B 0.000,C 90.000,E1 223.218} C_DIS
LIN {X -0.254,Y -559.604,Z 320.031,A 0.000,B 0.000,C 90.000,E1 221.595} C_DIS
LIN {X 0.097,Y -555.346,Z 320.023,A 0.000,B 0.000,C 90.000,E1 220.172} C_DIS
LIN {X 0.056,Y -549.324,Z 320.012,A 0.000,B 0.000,C 90.000,E1 218.222} C_DIS
LIN {X 0.301,Y -545.178,Z 320.005,A 0.000,B 0.000,C 90.000,E1 216.790} C_DIS
LIN {X -0.057,Y -537.069,Z 319.989,A 0.000,B 0.000,C 90.000,E1 213.992} C_DIS
LIN {X -0.208,Y -531.805,Z 319.978,A 0.000,B 0.000,C 90.000,E1 212.005} C_DIS
LIN {X 0.091,Y -526.040,Z 319.965,A 0.000,B 0.000,C 90.000,E1 209.667} C_DIS
LIN {X 0.023,Y -521.090,Z 319.954,A 0.000,B 0.000,C 90.000,E1 207.641} C_DIS
LIN {X 0.049,Y -516.300,Z 319.942,A 0.000,B 0.000,C 90.000,E1 205.591} C_DIS
LIN {X -0.039,Y -513.093,Z 319.934,A 0.000,B 0.000,C 90.000,E1 204.131} C_DIS
LIN {X 0.071,Y -509.791,Z 319.926,A 0.000,B 0.000,C 90.000,E1 202.642} C_DIS
LIN {X 0.119,Y -506.493,Z 319.918,A 0.000,B 0.000,C 90.000,E1 201.153} C_DIS
LIN {X -0.085,Y -502.036,Z 319.906,A 0.000,B 0.000,C 90.000,E1 199.087} C_DIS
LIN {X -0.025,Y -497.129,Z 319.893,A 0.000,B 0.000,C 90.000,E1 196.677} C_DIS
LIN {X 0.286,Y -493.683,Z 319.883,A 0.000,B 0.000,C 90.000,E1 194.828} C_DIS
LIN {X 0.167,Y -490.070,Z 319.871,A 0.000,B 0.000,C 90.000,E1 192.715} C_DIS
LIN {X -0.040,Y -486.487,Z 319.859,A 0.000,B 0.000,C 90.000,E1 190.602} C_DIS
LIN {X 0.159,Y -482.156,Z 319.844,A 0.000,B 0.000,C 90.000,E1 187.814} C_DIS
LIN {X 0.228,Y -478.693,Z 319.830,A 0.000,B 0.000,C 90.000,E1 185.334} C_DIS
LIN {X 0.165,Y -474.908,Z 319.813,A 0.000,B 0.000,C 90.000,E1 182.236} C_DIS
LIN {X 0.010,Y -470.852,Z 319.788,A 0.000,B 0.000,C 90.000,E1 177.879} C_DIS
LIN {X 0.183,Y -468.898,Z 319.767,A 0.000,B 0.000,C 90.000,E1 174.090} C_DIS
LIN {X 0.049,Y -468.288,Z 319.746,A 0.000,B 0.000,C 90.000,E1 170.330} C_DIS
LIN {X -0.141,Y -468.679,Z 319.731,A 0.000,B 0.000,C 90.000,E1 167.521} C_DIS
LIN {X 0.175,Y -469.914,Z 319.713,A 0.000,B 0.000,C 90.000,E1 164.338} C_DIS
LIN {X 0.085,Y -470.764,Z 319.704,A 0.000,B 0.000,C 90.000,E1 162.779} C_DIS
LIN {X 0.134,Y -472.867,Z 319.689,A 0.000,B 0.000,C 90.000,E1 159.953} C_DIS
LIN {X -0.011,Y -476.567,Z 319.670,A 0.000,B 0.000,C 90.000,E1 156.538} C_DIS
LIN {X -0.037,Y -482.114,Z 319.649,A 0.000,B 0.000,C 90.000,E1 152.820} C_DIS
LIN {X 0.028,Y -489.072,Z 319.629,A 0.000,B 0.000,C 90.000,E1 149.125} C_DIS
LIN {X -0.137,Y -494.695,Z 319.615,A 0.000,B 0.000,C 90.000,E1 146.707} C_DIS
LIN {X -0.013,Y -500.526,Z 319.602,A 0.000,B 0.000,C 90.000,E1 144.276} C_DIS
LIN {X 0.094,Y -504.108,Z 319.593,A 0.000,B 0.000,C 90.000,E1 142.763} C_DIS
LIN {X -0.023,Y -506.830,Z 319.587,A 0.000,B 0.000,C 90.000,E1 141.582} C_DIS
LIN {X 0.296,Y -509.211,Z 319.580,A 0.000,B 0.000,C 90.000,E1 140.356} C_DIS
LIN {X -0.141,Y -511.392,Z 319.573,A 0.000,B 0.000,C 90.000,E1 139.218} C_DIS
LIN {X -0.075,Y -512.863,Z 319.568,A 0.000,B 0.000,C 90.000,E1 138.324} C_DIS
LIN {X -0.119,Y -514.332,Z 319.562,A 0.000,B 0.000,C 90.000,E1 137.148} C_DIS
LIN {X -0.052,Y -515.104,Z 319.557,A 0.000,B 0.000,C 90.000,E1 136.257} C_DIS
LIN {X 0.035,Y -515.615,Z 319.552,A 0.000,B 0.000,C 90.000,E1 135.364} C_DIS
LIN {X -0.249,Y -515.752,Z 319.547,A 0.000,B 0.000,C 90.000,E1 134.514} C_DIS
LIN {X 0.102,Y -515.549,Z 319.541,A 0.000,B 0.000,C 90.000,E1 133.299} C_DIS
LIN {X -0.175,Y -515.049,Z 319.536,A 0.000,B 0.000,C 90.000,E1 132.447} C_DIS
LIN {X -0.070,Y -514.350,Z 319.531,A 0.000,B 0.000,C 90.000,E1 131.553} C_DIS
LIN {X -0.102,Y -512.997,Z 319.524,A 0.000,B 0.000,C 90.000,E1 130.378} C_DIS
LIN {X -0.101,Y -511.477,Z 319.518,A 0.000,B 0.000,C 90.000,E1 129.197} C_DIS
LIN {X -0.210,Y -509.334,Z 319.510,A 0.000,B 0.000,C 90.000,E1 127.729} C_DIS
LIN {X 0.137,Y -507.661,Z 319.503,A 0.000,B 0.000,C 90.000,E1 126.503} C_DIS
LIN {X 0.157,Y -505.853,Z 319.496,A 0.000,B 0.000,C 90.000,E1 125.311} C_DIS
LIN {X 0.037,Y -503.177,Z 319.488,A 0.000,B 0.000,C 90.000,E1 123.833} C_DIS
LIN {X 0.129,Y -500.816,Z 319.481,A 0.000,B 0.000,C 90.000,E1 122.625} C_DIS
LIN {X -0.231,Y -498.445,Z 319.475,A 0.000,B 0.000,C 90.000,E1 121.465} C_DIS
LIN {X 0.099,Y -494.698,Z 319.465,A 0.000,B 0.000,C 90.000,E1 119.617} C_DIS
LIN {X -0.095,Y -490.976,Z 319.455,A 0.000,B 0.000,C 90.000,E1 117.820} C_DIS
LIN {X 0.014,Y -487.829,Z 319.446,A 0.000,B 0.000,C 90.000,E1 116.283} C_DIS
LIN {X -0.134,Y -484.051,Z 319.436,A 0.000,B 0.000,C 90.000,E1 114.463} C_DIS
LIN {X 0.080,Y -479.485,Z 319.424,A 0.000,B 0.000,C 90.000,E1 112.280} C_DIS
LIN {X 0.026,Y -476.304,Z 319.415,A 0.000,B 0.000,C 90.000,E1 110.737} C_DIS
LIN {X -0.255,Y -473.055,Z 319.407,A 0.000,B 0.000,C 90.000,E1 109.214} C_DIS
LIN {X 0.053,Y -468.441,Z 319.394,A 0.000,B 0.000,C 90.000,E1 106.985} C_DIS
LIN {X 0.070,Y -465.697,Z 319.388,A 0.000,B 0.000,C 90.000,E1 105.733} C_DIS
LIN {X 0.156,Y -465.707,Z 319.387,A 0.000,B 0.000,C 90.000,E1 105.717} C_DIS
LIN {X 0.221,Y -467.572,Z 319.383,A 0.000,B 0.000,C 90.000,E1 104.954} C_DIS
LIN {X -0.047,Y -468.580,Z 319.380,A 0.000,B 0.000,C 90.000,E1 104.356} C_DIS
LIN {X 0.180,Y -475.805,Z 319.357,A 0.000,B 0.000,C 90.000,E1 100.254} C_DIS
LIN {X 0.018,Y -476.307,Z 319.355,A 0.000,B 0.000,C 90.000,E1 99.962} C_DIS
LIN {X -0.035,Y -481.792,Z 319.331,A 0.000,B 0.000,C 90.000,E1 95.625} C_DIS
LIN {X -0.188,Y -482.172,Z 319.330,A 0.000,B 0.000,C 90.000,E1 95.334} C_DIS
LIN {X 0.227,Y -485.310,Z 319.306,A 0.000,B 0.000,C 90.000,E1 90.974} C_DIS
LIN {X 0.051,Y -485.537,Z 319.304,A 0.000,B 0.000,C 90.000,E1 90.688} C_DIS
LIN {X -0.227,Y -486.320,Z 319.282,A 0.000,B 0.000,C 90.000,E1 86.731} C_DIS
LIN {X -0.092,Y -486.303,Z 319.278,A 0.000,B 0.000,C 90.000,E1 86.102} C_DIS
LIN {X 0.113,Y -484.696,Z 319.254,A 0.000,B 0.000,C 90.000,E1 81.781} C_DIS
LIN {X -0.019,Y -484.598,Z 319.253,A 0.000,B 0.000,C 90.000,E1 81.489} C_DIS
LIN {X -0.139,Y -480.532,Z 319.227,A 0.000,B 0.000,C 90.000,E1 76.881} C_DIS
LIN {X -0.215,Y -476.779,Z 319.213,A 0.000,B 0.000,C 90.000,E1 74.393} C_DIS
LIN {X 0.203,Y -476.781,Z 319.213,A 0.000,B 0.000,C 90.000,E1 74.338} C_DIS
LIN {X 0.006,Y -480.675,Z 319.205,A 0.000,B 0.000,C 90.000,E1 72.834} C_DIS
LIN {X -0.011,Y -486.369,Z 319.193,A 0.000,B 0.000,C 90.000,E1 70.678} C_DIS
LIN {X -0.028,Y -492.210,Z 319.181,A 0.000,B 0.000,C 90.000,E1 68.539} C_DIS
LIN {X -0.226,Y -497.299,Z 319.171,A 0.000,B 0.000,C 90.000,E1 66.741} C_DIS
LIN {X -0.112,Y -502.431,Z 319.161,A 0.000,B 0.000,C 90.000,E1 64.921} C_DIS
LIN {X 0.251,Y -506.769,Z 319.152,A 0.000,B 0.000,C 90.000,E1 63.384} C_DIS
LIN {X 0.231,Y -512.787,Z 319.141,A 0.000,B 0.000,C 90.000,E1 61.307} C_DIS
LIN {X -0.114,Y -517.057,Z 319.133,A 0.000,B 0.000,C 90.000,E1 59.871} C_DIS
LIN {X -0.194,Y -522.196,Z 319.123,A 0.000,B 0.000,C 90.000,E1 58.122} C_DIS
LIN {X -0.199,Y -528.048,Z 319.112,A 0.000,B 0.000,C 90.000,E1 56.087} C_DIS
LIN {X 0.123,Y -532.019,Z 319.104,A 0.000,B 0.000,C 90.000,E1 54.609} C_DIS
LIN {X -0.223,Y -535.065,Z 319.097,A 0.000,B 0.000,C 90.000,E1 53.497} C_DIS
LIN {X -0.216,Y -537.851,Z 319.091,A 0.000,B 0.000,C 90.000,E1 52.351} C_DIS
LIN {X 0.165,Y -540.385,Z 319.084,A 0.000,B 0.000,C 90.000,E1 51.170} C_DIS
LIN {X -0.198,Y -542.214,Z 319.080,A 0.000,B 0.000,C 90.000,E1 50.356} C_DIS
LIN {X -0.165,Y -544.329,Z 319.073,A 0.000,B 0.000,C 90.000,E1 49.218} C_DIS
LIN {X -0.101,Y -546.307,Z 319.067,A 0.000,B 0.000,C 90.000,E1 48.081} C_DIS
LIN {X -0.045,Y -547.563,Z 319.062,A 0.000,B 0.000,C 90.000,E1 47.229} C_DIS
LIN {X 0.066,Y -549.411,Z 319.055,A 0.000,B 0.000,C 90.000,E1 45.810} C_DIS
LIN {X 0.175,Y -550.439,Z 319.048,A 0.000,B 0.000,C 90.000,E1 44.676} C_DIS
LIN {X -0.125,Y -551.065,Z 319.044,A 0.000,B 0.000,C 90.000,E1 43.866} C_DIS
LIN {X -0.019,Y -551.544,Z 319.039,A 0.000,B 0.000,C 90.000,E1 43.014} C_DIS
LIN {X -0.264,Y -551.982,Z 319.033,A 0.000,B 0.000,C 90.000,E1 41.919} C_DIS
LIN {X -0.091,Y -552.060,Z 319.027,A 0.000,B 0.000,C 90.000,E1 40.782} C_DIS
LIN {X 0.022,Y -551.907,Z 319.022,A 0.000,B 0.000,C 90.000,E1 39.930} C_DIS
LIN {X -0.104,Y -551.219,Z 319.014,A 0.000,B 0.000,C 90.000,E1 38.543} C_DIS
LIN {X -0.240,Y -550.186,Z 319.006,A 0.000,B 0.000,C 90.000,E1 37.156} C_DIS
LIN {X -0.016,Y -549.131,Z 319.000,A 0.000,B 0.000,C 90.000,E1 36.011} C_DIS
LIN {X -0.079,Y -547.715,Z 318.992,A 0.000,B 0.000,C 90.000,E1 34.612} C_DIS
LIN {X 0.063,Y -545.699,Z 318.981,A 0.000,B 0.000,C 90.000,E1 32.625} C_DIS
LIN {X -0.138,Y -543.794,Z 318.970,A 0.000,B 0.000,C 90.000,E1 30.669} C_DIS
LIN {X 0.282,Y -541.769,Z 318.958,A 0.000,B 0.000,C 90.000,E1 28.359} C_DIS
LIN {X -0.096,Y -539.921,Z 318.947,A 0.000,B 0.000,C 90.000,E1 26.411} C_DIS
LIN {X 0.030,Y -538.621,Z 318.939,A 0.000,B 0.000,C 90.000,E1 24.975} C_DIS
LIN {X 0.301,Y -536.874,Z 318.928,A 0.000,B 0.000,C 90.000,E1 22.950} C_DIS
LIN {X -0.113,Y -535.578,Z 318.918,A 0.000,B 0.000,C 90.000,E1 21.280} C_DIS
LIN {X 0.163,Y -534.191,Z 318.905,A 0.000,B 0.000,C 90.000,E1 18.960} C_DIS
LIN {X -0.169,Y -533.310,Z 318.896,A 0.000,B 0.000,C 90.000,E1 17.275} C_DIS
LIN {X 0.024,Y -532.511,Z 318.885,A 0.000,B 0.000,C 90.000,E1 15.245} C_DIS
LIN {X -0.073,Y -531.936,Z 318.874,A 0.000,B 0.000,C 90.000,E1 13.244} C_DIS
LIN {X -0.100,Y -531.650,Z 318.859,A 0.000,B 0.000,C 90.000,E1 10.658} C_DIS
LIN {X 0.054,Y -531.745,Z 318.850,A 0.000,B 0.000,C 90.000,E1 8.916} C_DIS
LIN {X 0.135,Y -532.060,Z 318.840,A 0.000,B 0.000,C 90.000,E1 7.182} C_DIS
LIN {X 0.167,Y -532.653,Z 318.830,A 0.000,B 0.000,C 90.000,E1 5.454} C_DIS
LIN {X 0.211,Y -533.937,Z 318.816,A 0.000,B 0.000,C 90.000,E1 2.865} C_DIS
LIN {X 0.207,Y -535.165,Z 318.805,A 0.000,B 0.000,C 90.000,E1 0.859} C_DIS
LIN {X 0.256,Y -537.514,Z 318.788,A 0.000,B 0.000,C 90.000,E1 357.764} C_DIS
LIN {X -0.203,Y -539.292,Z 318.778,A 0.000,B 0.000,C 90.000,E1 356.102} C_DIS
LIN {X -0.084,Y -540.431,Z 318.772,A 0.000,B 0.000,C 90.000,E1 354.951} C_DIS
LIN {X 0.066,Y -541.990,Z 318.764,A 0.000,B 0.000,C 90.000,E1 353.514} C_DIS
LIN {X -0.133,Y -548.467,Z 318.744,A 0.000,B 0.000,C 90.000,E1 349.859} C_DIS
LIN {X -0.128,Y -552.042,Z 318.734,A 0.000,B 0.000,C 90.000,E1 348.173} C_DIS
LIN {X 0.174,Y -559.336,Z 318.719,A 0.000,B 0.000,C 90.000,E1 345.353} C_DIS
LIN {X 0.014,Y -564.835,Z 318.708,A 0.000,B 0.000,C 90.000,E1 343.433} C_DIS
LIN {X 0.208,Y -569.657,Z 318.699,A 0.000,B 0.000,C 90.000,E1 341.764} C_DIS
LIN {X -0.040,Y -573.778,Z 318.691,A 0.000,B 0.000,C 90.000,E1 340.423} C_DIS
LIN {X 0.165,Y -578.709,Z 318.682,A 0.000,B 0.000,C 90.000,E1 338.773} C_DIS
LIN {X 0.200,Y -585.784,Z 318.670,A 0.000,B 0.000,C 90.000,E1 336.613} C_DIS
LIN {X 0.254,Y -589.326,Z 318.664,A 0.000,B 0.000,C 90.000,E1 335.537} C_DIS
LIN {X 0.010,Y -594.022,Z 318.657,A 0.000,B 0.000,C 90.000,E1 334.229} C_DIS
LIN {X 0.281,Y -599.756,Z 318.648,A 0.000,B 0.000,C 90.000,E1 332.615} C_DIS
LIN {X 0.148,Y -605.305,Z 318.639,A 0.000,B 0.000,C 90.000,E1 331.051} C_DIS
LIN {X 0.119,Y -610.938,Z 318.631,A 0.000,B 0.000,C 90.000,E1 329.488} C_DIS
LIN {X 0.016,Y -615.650,Z 318.623,A 0.000,B 0.000,C 90.000,E1 328.201} C_DIS
LIN {X -0.004,Y -620.211,Z 318.616,A 0.000,B 0.000,C 90.000,E1 326.914} C_DIS
LIN {X -0.139,Y -625.317,Z 318.608,A 0.000,B 0.000,C 90.000,E1 325.388} C_DIS
LIN {X -0.163,Y -629.264,Z 318.601,A 0.000,B 0.000,C 90.000,E1 324.116} C_DIS
LIN {X -0.122,Y -632.971,Z 318.594,A 0.000,B 0.000,C 90.000,E1 322.844} C_DIS
LIN {X -0.017,Y -635.792,Z 318.588,A 0.000,B 0.000,C 90.000,E1 321.823} C_DIS
LIN {X -0.094,Y -640.825,Z 318.578,A 0.000,B 0.000,C 90.000,E1 320.070} C_DIS
LIN {X -0.063,Y -645.167,Z 318.570,A 0.000,B 0.000,C 90.000,E1 318.566} C_DIS
LIN {X -0.106,Y -650.999,Z 318.559,A 0.000,B 0.000,C 90.000,E1 316.581} C_DIS
LIN {X 0.129,Y -654.919,Z 318.552,A 0.000,B 0.000,C 90.000,E1 315.324} C_DIS
LIN {X -0.071,Y -659.253,Z 318.544,A 0.000,B 0.000,C 90.000,E1 313.866} C_DIS
LIN {X 0.319,Y -662.059,Z 318.538,A 0.000,B 0.000,C 90.000,E1 312.852} C_DIS
LIN {X -0.202,Y -665.267,Z 318.531,A 0.000,B 0.000,C 90.000,E1 311.676} C_DIS
LIN {X -0.181,Y -668.277,Z 318.525,A 0.000,B 0.000,C 90.000,E1 310.458} C_DIS
LIN {X -0.024,Y -671.568,Z 318.517,A 0.000,B 0.000,C 90.000,E1 308.991} C_DIS
LIN {X -0.333,Y -673.975,Z 318.510,A 0.000,B 0.000,C 90.000,E1 307.810} C_DIS
LIN {X -0.208,Y -675.245,Z 318.506,A 0.000,B 0.000,C 90.000,E1 307.076} C_DIS
LIN {X -0.076,Y -676.359,Z 318.502,A 0.000,B 0.000,C 90.000,E1 306.343} C_DIS
LIN {X 0.213,Y -677.270,Z 318.498,A 0.000,B 0.000,C 90.000,E1 305.598} C_DIS
LIN {X -0.031,Y -677.968,Z 318.494,A 0.000,B 0.000,C 90.000,E1 304.898} C_DIS
LIN {X -0.270,Y -678.464,Z 318.490,A 0.000,B 0.000,C 90.000,E1 304.199} C_DIS
LIN {X -0.114,Y -678.678,Z 318.487,A 0.000,B 0.000,C 90.000,E1 303.706} C_DIS
LIN {X -0.176,Y -678.700,Z 318.482,A 0.000,B 0.000,C 90.000,E1 302.752} C_DIS
LIN {X 0.156,Y -678.443,Z 318.478,A 0.000,B 0.000,C 90.000,E1 302.005} C_DIS
LIN {X -0.448,Y -677.904,Z 318.474,A 0.000,B 0.000,C 90.000,E1 301.337} C_DIS
LIN {X -0.128,Y -677.057,Z 318.470,A 0.000,B 0.000,C 90.000,E1 300.590} C_DIS
LIN {X -0.161,Y -675.911,Z 318.466,A 0.000,B 0.000,C 90.000,E1 299.873} C_DIS
LIN {X -0.017,Y -674.096,Z 318.461,A 0.000,B 0.000,C 90.000,E1 298.899} C_DIS
LIN {X -0.313,Y -671.354,Z 318.454,A 0.000,B 0.000,C 90.000,E1 297.719} C_DIS
LIN {X -0.066,Y -668.441,Z 318.447,A 0.000,B 0.000,C 90.000,E1 296.488} C_DIS
LIN {X -0.015,Y -664.598,Z 318.439,A 0.000,B 0.000,C 90.000,E1 295.027} C_DIS
LIN {X -0.049,Y -660.683,Z 318.431,A 0.000,B 0.000,C 90.000,E1 293.567} C_DIS
LIN {X 0.039,Y -655.927,Z 318.421,A 0.000,B 0.000,C 90.000,E1 291.844} C_DIS
LIN {X 0.026,Y -651.268,Z 318.412,A 0.000,B 0.000,C 90.000,E1 290.120} C_DIS
LIN {X 0.291,Y -646.866,Z 318.402,A 0.000,B 0.000,C 90.000,E1 288.362} C_DIS
LIN {X -0.207,Y -643.326,Z 318.394,A 0.000,B 0.000,C 90.000,E1 286.913} C_DIS
LIN {X -0.213,Y -637.992,Z 318.380,A 0.000,B 0.000,C 90.000,E1 284.411} C_DIS
LIN {X 0.282,Y -631.884,Z 318.360,A 0.000,B 0.000,C 90.000,E1 280.838} C_DIS
LIN {X -0.133,Y -628.708,Z 318.346,A 0.000,B 0.000,C 90.000,E1 278.341} C_DIS
LIN {X -0.214,Y -625.572,Z 318.325,A 0.000,B 0.000,C 90.000,E1 274.531} C_DIS
LIN {X 0.109,Y -624.593,Z 318.311,A 0.000,B 0.000,C 90.000,E1 271.949} C_DIS
LIN {X 0.049,Y -624.371,Z 318.298,A 0.000,B 0.000,C 90.000,E1 269.656} C_DIS
LIN {X -0.014,Y -624.818,Z 318.285,A 0.000,B 0.000,C 90.000,E1 267.364} C_DIS
LIN {X 0.115,Y -625.309,Z 318.280,A 0.000,B 0.000,C 90.000,E1 266.331} C_DIS
LIN {X -0.081,Y -626.936,Z 318.266,A 0.000,B 0.000,C 90.000,E1 263.799} C_DIS
LIN {X -0.068,Y -629.229,Z 318.251,A 0.000,B 0.000,C 90.000,E1 261.254} C_DIS
LIN {X -0.006,Y -631.511,Z 318.240,A 0.000,B 0.000,C 90.000,E1 259.218} C_DIS
LIN {X -0.126,Y -634.925,Z 318.226,A 0.000,B 0.000,C 90.000,E1 256.700} C_DIS
LIN {X 0.227,Y -636.688,Z 318.219,A 0.000,B 0.000,C 90.000,E1 255.408} C_DIS
LIN {X 0.323,Y -637.966,Z 318.214,A 0.000,B 0.000,C 90.000,E1 254.393} C_DIS
LIN {X 0.103,Y -639.335,Z 318.205,A 0.000,B 0.000,C 90.000,E1 252.906} C_DIS
LIN {X -0.379,Y -640.128,Z 318.200,A 0.000,B 0.000,C 90.000,E1 251.945} C_DIS
LIN {X -0.041,Y -640.671,Z 318.194,A 0.000,B 0.000,C 90.000,E1 250.913} C_DIS
LIN {X -0.169,Y -640.763,Z 318.191,A 0.000,B 0.000,C 90.000,E1 250.423} C_DIS
LIN {X 0.178,Y -640.536,Z 318.186,A 0.000,B 0.000,C 90.000,E1 249.390} C_DIS
LIN {X 0.102,Y -640.201,Z 318.181,A 0.000,B 0.000,C 90.000,E1 248.646} C_DIS
LIN {X -0.215,Y -639.464,Z 318.177,A 0.000,B 0.000,C 90.000,E1 247.922} C_DIS
LIN {X -0.303,Y -638.498,Z 318.173,A 0.000,B 0.000,C 90.000,E1 247.177} C_DIS
LIN {X -0.351,Y -636.769,Z 318.168,A 0.000,B 0.000,C 90.000,E1 246.177} C_DIS
LIN {X -0.157,Y -634.679,Z 318.162,A 0.000,B 0.000,C 90.000,E1 245.153} C_DIS
LIN {X -0.337,Y -633.501,Z 318.159,A 0.000,B 0.000,C 90.000,E1 244.665} C_DIS
LIN {X -0.219,Y -631.470,Z 318.155,A 0.000,B 0.000,C 90.000,E1 243.896} C_DIS
LIN {X -0.066,Y -627.713,Z 318.148,A 0.000,B 0.000,C 90.000,E1 242.615} C_DIS
LIN {X -0.222,Y -622.160,Z 318.138,A 0.000,B 0.000,C 90.000,E1 240.845} C_DIS
LIN {X 0.061,Y -618.099,Z 318.131,A 0.000,B 0.000,C 90.000,E1 239.537} C_DIS
LIN {X 0.020,Y -613.180,Z 318.122,A 0.000,B 0.000,C 90.000,E1 237.995} C_DIS
LIN {X -0.070,Y -609.086,Z 318.115,A 0.000,B 0.000,C 90.000,E1 236.707} C_DIS
LIN {X 0.106,Y -604.896,Z 318.108,A 0.000,B 0.000,C 90.000,E1 235.388} C_DIS
LIN {X 0.205,Y -600.728,Z 318.101,A 0.000,B 0.000,C 90.000,E1 234.069} C_DIS
LIN {X -0.137,Y -597.220,Z 318.095,A 0.000,B 0.000,C 90.000,E1 233.050} C_DIS
LIN {X -0.072,Y -591.663,Z 318.086,A 0.000,B 0.000,C 90.000,E1 231.457} C_DIS
LIN {X 0.242,Y -586.252,Z 318.077,A 0.000,B 0.000,C 90.000,E1 229.828} C_DIS
LIN {X -0.117,Y -579.233,Z 318.065,A 0.000,B 0.000,C 90.000,E1 227.715} C_DIS
LIN {X -0.265,Y -575.016,Z 318.058,A 0.000,B 0.000,C 90.000,E1 226.377} C_DIS
LIN {X 0.208,Y -571.448,Z 318.052,A 0.000,B 0.000,C 90.000,E1 225.243} C_DIS
LIN {X 0.115,Y -565.454,Z 318.041,A 0.000,B 0.000,C 90.000,E1 223.338} C_DIS
LIN {X -0.263,Y -561.229,Z 318.033,A 0.000,B 0.000,C 90.000,E1 222.000} C_DIS
LIN {X 0.140,Y -556.101,Z 318.024,A 0.000,B 0.000,C 90.000,E1 220.297} C_DIS
LIN {X 0.136,Y -550.920,Z 318.015,A 0.000,B 0.000,C 90.000,E1 218.624} C_DIS
LIN {X -0.015,Y -546.813,Z 318.007,A 0.000,B 0.000,C 90.000,E1 217.237} C_DIS
LIN {X -0.014,Y -539.386,Z 317.993,A 0.000,B 0.000,C 90.000,E1 214.692} C_DIS
LIN {X 0.187,Y -533.990,Z 317.982,A 0.000,B 0.000,C 90.000,E1 212.673} C_DIS
LIN {X -0.002,Y -530.299,Z 317.974,A 0.000,B 0.000,C 90.000,E1 211.258} C_DIS
LIN {X -0.112,Y -525.952,Z 317.964,A 0.000,B 0.000,C 90.000,E1 209.539} C_DIS
LIN {X -0.179,Y -520.985,Z 317.953,A 0.000,B 0.000,C 90.000,E1 207.513} C_DIS
LIN {X -0.235,Y -514.262,Z 317.937,A 0.000,B 0.000,C 90.000,E1 204.591} C_DIS
LIN {X 0.222,Y -510.327,Z 317.927,A 0.000,B 0.000,C 90.000,E1 202.770} C_DIS
LIN {X -0.274,Y -506.378,Z 317.917,A 0.000,B 0.000,C 90.000,E1 201.046} C_DIS
LIN {X 0.093,Y -502.616,Z 317.907,A 0.000,B 0.000,C 90.000,E1 199.214} C_DIS
LIN {X 0.177,Y -497.736,Z 317.894,A 0.000,B 0.000,C 90.000,E1 196.804} C_DIS
LIN {X -0.005,Y -494.902,Z 317.885,A 0.000,B 0.000,C 90.000,E1 195.315} C_DIS
LIN {X -0.065,Y -490.233,Z 317.870,A 0.000,B 0.000,C 90.000,E1 192.591} C_DIS
LIN {X 0.114,Y -486.668,Z 317.858,A 0.000,B 0.000,C 90.000,E1 190.433} C_DIS
LIN {X -0.150,Y -482.398,Z 317.843,A 0.000,B 0.000,C 90.000,E1 187.701} C_DIS
LIN {X -0.066,Y -478.946,Z 317.829,A 0.000,B 0.000,C 90.000,E1 185.220} C_DIS
LIN {X 0.095,Y -475.572,Z 317.813,A 0.000,B 0.000,C 90.000,E1 182.407} C_DIS
LIN {X 0.225,Y -471.269,Z 317.787,A 0.000,B 0.000,C 90.000,E1 177.707} C_DIS
LIN {X -0.008,Y -469.411,Z 317.767,A 0.000,B 0.000,C 90.000,E1 173.970} C_DIS
LIN {X -0.096,Y -468.839,Z 317.746,A 0.000,B 0.000,C 90.000,E1 170.208} C_DIS
LIN {X 0.104,Y -469.229,Z 317.730,A 0.000,B 0.000,C 90.000,E1 167.353} C_DIS
LIN {X 0.099,Y -470.490,Z 317.712,A 0.000,B 0.000,C 90.000,E1 164.212} C_DIS
LIN {X 0.072,Y -471.179,Z 317.705,A 0.000,B 0.000,C 90.000,E1 162.960} C_DIS
LIN {X 0.100,Y -473.452,Z 317.688,A 0.000,B 0.000,C 90.000,E1 159.826} C_DIS
LIN {X -0.014,Y -477.165,Z 317.669,A 0.000,B 0.000,C 90.000,E1 156.410} C_DIS
LIN {X -0.012,Y -482.704,Z 317.648,A 0.000,B 0.000,C 90.000,E1 152.692} C_DIS
LIN {X -0.166,Y -488.932,Z 317.630,A 0.000,B 0.000,C 90.000,E1 149.331} C_DIS
LIN {X -0.070,Y -494.353,Z 317.616,A 0.000,B 0.000,C 90.000,E1 146.882} C_DIS
LIN {X -0.230,Y -500.002,Z 317.603,A 0.000,B 0.000,C 90.000,E1 144.482} C_DIS
LIN {X -0.076,Y -501.398,Z 317.599,A 0.000,B 0.000,C 90.000,E1 143.863} C_DIS
LIN {X 0.156,Y -504.157,Z 317.593,A 0.000,B 0.000,C 90.000,E1 142.637} C_DIS
LIN {X 0.035,Y -506.754,Z 317.586,A 0.000,B 0.000,C 90.000,E1 141.457} C_DIS
LIN {X 0.052,Y -508.488,Z 317.581,A 0.000,B 0.000,C 90.000,E1 140.561} C_DIS
LIN {X -0.003,Y -510.625,Z 317.574,A 0.000,B 0.000,C 90.000,E1 139.380} C_DIS
LIN {X 0.053,Y -512.085,Z 317.569,A 0.000,B 0.000,C 90.000,E1 138.485} C_DIS
LIN {X -0.004,Y -513.549,Z 317.563,A 0.000,B 0.000,C 90.000,E1 137.310} C_DIS
LIN {X 0.053,Y -514.331,Z 317.558,A 0.000,B 0.000,C 90.000,E1 136.419} C_DIS
LIN {X -0.235,Y -514.872,Z 317.553,A 0.000,B 0.000,C 90.000,E1 135.567} C_DIS
LIN {X 0.108,Y -515.041,Z 317.547,A 0.000,B 0.000,C 90.000,E1 134.352} C_DIS
LIN {X 0.181,Y -514.908,Z 317.542,A 0.000,B 0.000,C 90.000,E1 133.461} C_DIS
LIN {X -0.101,Y -514.465,Z 317.537,A 0.000,B 0.000,C 90.000,E1 132.609} C_DIS
LIN {X -0.003,Y -513.790,Z 317.532,A 0.000,B 0.000,C 90.000,E1 131.714} C_DIS
LIN {X -0.041,Y -512.464,Z 317.525,A 0.000,B 0.000,C 90.000,E1 130.539} C_DIS
LIN {X 0.192,Y -510.545,Z 317.517,A 0.000,B 0.000,C 90.000,E1 129.036} C_DIS
LIN {X 0.061,Y -508.426,Z 317.509,A 0.000,B 0.000,C 90.000,E1 127.569} C_DIS
LIN {X 0.088,Y -506.737,Z 317.502,A 0.000,B 0.000,C 90.000,E1 126.377} C_DIS
LIN {X 0.098,Y -504.852,Z 317.496,A 0.000,B 0.000,C 90.000,E1 125.185} C_DIS
LIN {X -0.036,Y -502.141,Z 317.487,A 0.000,B 0.000,C 90.000,E1 123.706} C_DIS
LIN {X 0.045,Y -499.784,Z 317.481,A 0.000,B 0.000,C 90.000,E1 122.498} C_DIS
LIN {X -0.328,Y -497.393,Z 317.474,A 0.000,B 0.000,C 90.000,E1 121.337} C_DIS
LIN {X -0.044,Y -494.292,Z 317.466,A 0.000,B 0.000,C 90.000,E1 119.795} C_DIS
LIN {X 0.200,Y -489.951,Z 317.454,A 0.000,B 0.000,C 90.000,E1 117.641} C_DIS
LIN {X -0.144,Y -486.823,Z 317.445,A 0.000,B 0.000,C 90.000,E1 116.155} C_DIS
LIN {X 0.128,Y -483.066,Z 317.435,A 0.000,B 0.000,C 90.000,E1 114.283} C_DIS
LIN {X -0.117,Y -479.172,Z 317.425,A 0.000,B 0.000,C 90.000,E1 112.461} C_DIS
LIN {X -0.197,Y -475.387,Z 317.414,A 0.000,B 0.000,C 90.000,E1 110.610} C_DIS
LIN {X -0.050,Y -472.197,Z 317.406,A 0.000,B 0.000,C 90.000,E1 109.033} C_DIS
LIN {X -0.214,Y -467.753,Z 317.394,A 0.000,B 0.000,C 90.000,E1 106.858} C_DIS
LIN {X 0.084,Y -465.563,Z 317.388,A 0.000,B 0.000,C 90.000,E1 105.788} C_DIS
LIN {X 0.043,Y -465.571,Z 317.388,A 0.000,B 0.000,C 90.000,E1 105.788} C_DIS
LIN {X -0.114,Y -467.676,Z 317.383,A 0.000,B 0.000,C 90.000,E1 104.954} C_DIS
LIN {X -0.158,Y -475.890,Z 317.357,A 0.000,B 0.000,C 90.000,E1 100.254} C_DIS
LIN {X 0.149,Y -476.344,Z 317.355,A 0.000,B 0.000,C 90.000,E1 99.905} C_DIS
LIN {X 0.106,Y -481.857,Z 317.331,A 0.000,B 0.000,C 90.000,E1 95.568} C_DIS
LIN {X -0.046,Y -482.188,Z 317.329,A 0.000,B 0.000,C 90.000,E1 95.277} C_DIS
LIN {X -0.113,Y -485.352,Z 317.305,A 0.000,B 0.000,C 90.000,E1 90.974} C_DIS
LIN {X 0.197,Y -485.533,Z 317.304,A 0.000,B 0.000,C 90.000,E1 90.630} C_DIS
LIN {X -0.081,Y -486.340,Z 317.282,A 0.000,B 0.000,C 90.000,E1 86.674} C_DIS
LIN {X 0.054,Y -486.275,Z 317.278,A 0.000,B 0.000,C 90.000,E1 86.045} C_DIS
LIN {X -0.226,Y -484.694,Z 317.254,A 0.000,B 0.000,C 90.000,E1 81.781} C_DIS
LIN {X 0.122,Y -484.549,Z 317.253,A 0.000,B 0.000,C 90.000,E1 81.432} C_DIS
LIN {X -0.009,Y -480.488,Z 317.227,A 0.000,B 0.000,C 90.000,E1 76.825} C_DIS
LIN {X 0.065,Y -476.585,Z 317.212,A 0.000,B 0.000,C 90.000,E1 74.212} C_DIS
LIN {X 0.025,Y -476.585,Z 317.212,A 0.000,B 0.000,C 90.000,E1 74.212} C_DIS
LIN {X -0.043,Y -480.940,Z 317.203,A 0.000,B 0.000,C 90.000,E1 72.489} C_DIS
LIN {X 0.244,Y -485.766,Z 317.192,A 0.000,B 0.000,C 90.000,E1 70.604} C_DIS
LIN {X 0.192,Y -490.729,Z 317.182,A 0.000,B 0.000,C 90.000,E1 68.773} C_DIS
LIN {X -0.074,Y -494.968,Z 317.174,A 0.000,B 0.000,C 90.000,E1 67.283} C_DIS
LIN {X 0.189,Y -499.231,Z 317.165,A 0.000,B 0.000,C 90.000,E1 65.741} C_DIS
LIN {X 0.112,Y -504.428,Z 317.155,A 0.000,B 0.000,C 90.000,E1 63.948} C_DIS
LIN {X -0.163,Y -508.709,Z 317.147,A 0.000,B 0.000,C 90.000,E1 62.487} C_DIS
LIN {X 0.208,Y -513.880,Z 317.137,A 0.000,B 0.000,C 90.000,E1 60.667} C_DIS
LIN {X 0.060,Y -519.020,Z 317.127,A 0.000,B 0.000,C 90.000,E1 58.918} C_DIS
LIN {X 0.139,Y -522.439,Z 317.121,A 0.000,B 0.000,C 90.000,E1 57.740} C_DIS
LIN {X 0.020,Y -527.459,Z 317.111,A 0.000,B 0.000,C 90.000,E1 56.008} C_DIS
LIN {X 0.029,Y -531.439,Z 317.103,A 0.000,B 0.000,C 90.000,E1 54.562} C_DIS
LIN {X -0.014,Y -534.491,Z 317.097,A 0.000,B 0.000,C 90.000,E1 53.417} C_DIS
LIN {X -0.012,Y -537.282,Z 317.090,A 0.000,B 0.000,C 90.000,E1 52.271} C_DIS
LIN {X 0.024,Y -539.823,Z 317.084,A 0.000,B 0.000,C 90.000,E1 51.126} C_DIS
LIN {X -0.005,Y -541.628,Z 317.079,A 0.000,B 0.000,C 90.000,E1 50.275} C_DIS
LIN {X 0.046,Y -544.262,Z 317.071,A 0.000,B 0.000,C 90.000,E1 48.852} C_DIS
LIN {X 0.106,Y -546.138,Z 317.065,A 0.000,B 0.000,C 90.000,E1 47.715} C_DIS
LIN {X -0.215,Y -547.718,Z 317.059,A 0.000,B 0.000,C 90.000,E1 46.620} C_DIS
LIN {X 0.231,Y -548.786,Z 317.054,A 0.000,B 0.000,C 90.000,E1 45.729} C_DIS
LIN {X -0.061,Y -549.808,Z 317.048,A 0.000,B 0.000,C 90.000,E1 44.636} C_DIS
LIN {X 0.062,Y -550.590,Z 317.042,A 0.000,B 0.000,C 90.000,E1 43.500} C_DIS
LIN {X 0.182,Y -551.152,Z 317.036,A 0.000,B 0.000,C 90.000,E1 42.366} C_DIS
LIN {X -0.079,Y -551.432,Z 317.031,A 0.000,B 0.000,C 90.000,E1 41.553} C_DIS
LIN {X 0.089,Y -551.472,Z 317.025,A 0.000,B 0.000,C 90.000,E1 40.415} C_DIS
LIN {X 0.195,Y -551.259,Z 317.020,A 0.000,B 0.000,C 90.000,E1 39.564} C_DIS
LIN {X 0.001,Y -550.733,Z 317.014,A 0.000,B 0.000,C 90.000,E1 38.463} C_DIS
LIN {X -0.147,Y -549.737,Z 317.006,A 0.000,B 0.000,C 90.000,E1 37.076} C_DIS
LIN {X 0.017,Y -548.995,Z 317.001,A 0.000,B 0.000,C 90.000,E1 36.217} C_DIS
LIN {X -0.051,Y -547.628,Z 316.993,A 0.000,B 0.000,C 90.000,E1 34.818} C_DIS
LIN {X 0.051,Y -545.916,Z 316.984,A 0.000,B 0.000,C 90.000,E1 33.118} C_DIS
LIN {X -0.080,Y -544.543,Z 316.976,A 0.000,B 0.000,C 90.000,E1 31.720} C_DIS
LIN {X 0.118,Y -543.232,Z 316.968,A 0.000,B 0.000,C 90.000,E1 30.285} C_DIS
LIN {X 0.053,Y -541.468,Z 316.957,A 0.000,B 0.000,C 90.000,E1 28.309} C_DIS
LIN {X 0.206,Y -540.127,Z 316.949,A 0.000,B 0.000,C 90.000,E1 26.873} C_DIS
LIN {X -0.186,Y -538.571,Z 316.940,A 0.000,B 0.000,C 90.000,E1 25.207} C_DIS
LIN {X 0.076,Y -536.575,Z 316.927,A 0.000,B 0.000,C 90.000,E1 22.898} C_DIS
LIN {X 0.161,Y -535.277,Z 316.918,A 0.000,B 0.000,C 90.000,E1 21.173} C_DIS
LIN {X -0.063,Y -533.878,Z 316.905,A 0.000,B 0.000,C 90.000,E1 18.906} C_DIS
LIN {X -0.207,Y -532.822,Z 316.894,A 0.000,B 0.000,C 90.000,E1 16.913} C_DIS
LIN {X -0.207,Y -532.168,Z 316.884,A 0.000,B 0.000,C 90.000,E1 15.190} C_DIS
LIN {X -0.186,Y -531.588,Z 316.873,A 0.000,B 0.000,C 90.000,E1 13.175} C_DIS
LIN {X 0.182,Y -531.281,Z 316.859,A 0.000,B 0.000,C 90.000,E1 10.546} C_DIS
LIN {X -0.118,Y -531.438,Z 316.846,A 0.000,B 0.000,C 90.000,E1 8.276} C_DIS
LIN {X -0.074,Y -532.080,Z 316.832,A 0.000,B 0.000,C 90.000,E1 5.682} C_DIS
LIN {X -0.074,Y -533.086,Z 316.819,A 0.000,B 0.000,C 90.000,E1 3.383} C_DIS
LIN {X -0.073,Y -534.073,Z 316.809,A 0.000,B 0.000,C 90.000,E1 1.661} C_DIS
LIN {X 0.203,Y -535.217,Z 316.799,A 0.000,B 0.000,C 90.000,E1 359.771} C_DIS
LIN {X 0.255,Y -537.688,Z 316.783,A 0.000,B 0.000,C 90.000,E1 356.906} C_DIS
LIN {X -0.189,Y -538.852,Z 316.777,A 0.000,B 0.000,C 90.000,E1 355.812} C_DIS
LIN {X 0.078,Y -541.613,Z 316.762,A 0.000,B 0.000,C 90.000,E1 353.223} C_DIS
LIN {X -0.225,Y -547.627,Z 316.744,A 0.000,B 0.000,C 90.000,E1 349.859} C_DIS
LIN {X -0.240,Y -551.169,Z 316.734,A 0.000,B 0.000,C 90.000,E1 348.173} C_DIS
LIN {X -0.103,Y -557.647,Z 316.720,A 0.000,B 0.000,C 90.000,E1 345.644} C_DIS
LIN {X -0.065,Y -562.290,Z 316.711,A 0.000,B 0.000,C 90.000,E1 343.976} C_DIS
LIN {X -0.139,Y -567.867,Z 316.700,A 0.000,B 0.000,C 90.000,E1 342.054} C_DIS
LIN {X -0.063,Y -571.956,Z 316.693,A 0.000,B 0.000,C 90.000,E1 340.678} C_DIS
LIN {X 0.095,Y -576.912,Z 316.684,A 0.000,B 0.000,C 90.000,E1 339.028} C_DIS
LIN {X -0.063,Y -584.809,Z 316.670,A 0.000,B 0.000,C 90.000,E1 336.613} C_DIS
LIN {X -0.029,Y -593.077,Z 316.657,A 0.000,B 0.000,C 90.000,E1 334.204} C_DIS
LIN {X -0.038,Y -598.791,Z 316.648,A 0.000,B 0.000,C 90.000,E1 332.615} C_DIS
LIN {X -0.128,Y -603.431,Z 316.641,A 0.000,B 0.000,C 90.000,E1 331.307} C_DIS
LIN {X 0.065,Y -609.973,Z 316.630,A 0.000,B 0.000,C 90.000,E1 329.459} C_DIS
LIN {X -0.368,Y -614.640,Z 316.623,A 0.000,B 0.000,C 90.000,E1 328.201} C_DIS
LIN {X -0.069,Y -619.218,Z 316.616,A 0.000,B 0.000,C 90.000,E1 326.882} C_DIS
LIN {X -0.053,Y -624.363,Z 316.607,A 0.000,B 0.000,C 90.000,E1 325.341} C_DIS
LIN {X -0.100,Y -628.389,Z 316.600,A 0.000,B 0.000,C 90.000,E1 324.069} C_DIS
LIN {X 0.301,Y -632.140,Z 316.593,A 0.000,B 0.000,C 90.000,E1 322.763} C_DIS
LIN {X -0.117,Y -635.710,Z 316.586,A 0.000,B 0.000,C 90.000,E1 321.537} C_DIS
LIN {X -0.296,Y -641.514,Z 316.575,A 0.000,B 0.000,C 90.000,E1 319.542} C_DIS
LIN {X 0.251,Y -645.139,Z 316.568,A 0.000,B 0.000,C 90.000,E1 318.243} C_DIS
LIN {X -0.337,Y -652.531,Z 316.554,A 0.000,B 0.000,C 90.000,E1 315.810} C_DIS
LIN {X -0.008,Y -654.838,Z 316.550,A 0.000,B 0.000,C 90.000,E1 315.040} C_DIS
LIN {X 0.312,Y -657.731,Z 316.545,A 0.000,B 0.000,C 90.000,E1 314.028} C_DIS
LIN {X -0.274,Y -661.189,Z 316.538,A 0.000,B 0.000,C 90.000,E1 312.852} C_DIS
LIN {X 0.127,Y -664.392,Z 316.531,A 0.000,B 0.000,C 90.000,E1 311.595} C_DIS
LIN {X 0.134,Y -667.380,Z 316.524,A 0.000,B 0.000,C 90.000,E1 310.378} C_DIS
LIN {X 0.272,Y -670.610,Z 316.516,A 0.000,B 0.000,C 90.000,E1 308.910} C_DIS
LIN {X -0.049,Y -672.521,Z 316.511,A 0.000,B 0.000,C 90.000,E1 307.971} C_DIS
LIN {X -0.056,Y -673.465,Z 316.508,A 0.000,B 0.000,C 90.000,E1 307.488} C_DIS
LIN {X 0.188,Y -675.013,Z 316.503,A 0.000,B 0.000,C 90.000,E1 306.503} C_DIS
LIN {X -0.091,Y -676.224,Z 316.498,A 0.000,B 0.000,C 90.000,E1 305.564} C_DIS
LIN {X 0.204,Y -676.898,Z 316.494,A 0.000,B 0.000,C 90.000,E1 304.818} C_DIS
LIN {X 0.119,Y -677.500,Z 316.488,A 0.000,B 0.000,C 90.000,E1 303.865} C_DIS
LIN {X 0.020,Y -677.509,Z 316.482,A 0.000,B 0.000,C 90.000,E1 302.673} C_DIS
LIN {X -0.022,Y -677.226,Z 316.478,A 0.000,B 0.000,C 90.000,E1 301.957} C_DIS
LIN {X -0.281,Y -676.611,Z 316.474,A 0.000,B 0.000,C 90.000,E1 301.258} C_DIS
LIN {X 0.022,Y -675.720,Z 316.470,A 0.000,B 0.000,C 90.000,E1 300.512} C_DIS
LIN {X -0.025,Y -674.546,Z 316.466,A 0.000,B 0.000,C 90.000,E1 299.795} C_DIS
LIN {X -0.080,Y -673.195,Z 316.462,A 0.000,B 0.000,C 90.000,E1 299.077} C_DIS
LIN {X 0.196,Y -670.458,Z 316.455,A 0.000,B 0.000,C 90.000,E1 297.847} C_DIS
LIN {X -0.171,Y -667.546,Z 316.448,A 0.000,B 0.000,C 90.000,E1 296.668} C_DIS
LIN {X -0.292,Y -664.387,Z 316.441,A 0.000,B 0.000,C 90.000,E1 295.463} C_DIS
LIN {X 0.142,Y -661.119,Z 316.435,A 0.000,B 0.000,C 90.000,E1 294.207} C_DIS
LIN {X -0.335,Y -659.142,Z 316.431,A 0.000,B 0.000,C 90.000,E1 293.515} C_DIS
LIN {X -0.135,Y -655.054,Z 316.422,A 0.000,B 0.000,C 90.000,E1 292.025} C_DIS
LIN {X -0.254,Y -651.087,Z 316.414,A 0.000,B 0.000,C 90.000,E1 290.556} C_DIS
LIN {X 0.076,Y -645.988,Z 316.403,A 0.000,B 0.000,C 90.000,E1 288.544} C_DIS
LIN {X 0.023,Y -641.829,Z 316.393,A 0.000,B 0.000,C 90.000,E1 286.804} C_DIS
LIN {X -0.019,Y -636.531,Z 316.379,A 0.000,B 0.000,C 90.000,E1 284.300} C_DIS
LIN {X 0.116,Y -630.858,Z 316.361,A 0.000,B 0.000,C 90.000,E1 281.007} C_DIS
LIN {X 0.063,Y -627.356,Z 316.346,A 0.000,B 0.000,C 90.000,E1 278.219} C_DIS
LIN {X 0.127,Y -624.409,Z 316.326,A 0.000,B 0.000,C 90.000,E1 274.645} C_DIS
LIN {X -0.218,Y -623.415,Z 316.312,A 0.000,B 0.000,C 90.000,E1 272.121} C_DIS
LIN {X 0.309,Y -623.147,Z 316.299,A 0.000,B 0.000,C 90.000,E1 269.771} C_DIS
LIN {X -0.082,Y -623.641,Z 316.285,A 0.000,B 0.000,C 90.000,E1 267.249} C_DIS
LIN {X 0.111,Y -624.414,Z 316.276,A 0.000,B 0.000,C 90.000,E1 265.698} C_DIS
LIN {X 0.185,Y -626.021,Z 316.263,A 0.000,B 0.000,C 90.000,E1 263.394} C_DIS
LIN {X -0.241,Y -628.178,Z 316.251,A 0.000,B 0.000,C 90.000,E1 261.141} C_DIS
LIN {X -0.214,Y -630.499,Z 316.239,A 0.000,B 0.000,C 90.000,E1 259.106} C_DIS
LIN {X -0.196,Y -633.644,Z 316.227,A 0.000,B 0.000,C 90.000,E1 256.825} C_DIS
LIN {X 0.288,Y -635.449,Z 316.220,A 0.000,B 0.000,C 90.000,E1 255.519} C_DIS
LIN {X 0.202,Y -636.781,Z 316.214,A 0.000,B 0.000,C 90.000,E1 254.519} C_DIS
LIN {X 0.126,Y -637.965,Z 316.207,A 0.000,B 0.000,C 90.000,E1 253.268} C_DIS
LIN {X -0.374,Y -638.853,Z 316.202,A 0.000,B 0.000,C 90.000,E1 252.308} C_DIS
LIN {X -0.228,Y -639.642,Z 316.195,A 0.000,B 0.000,C 90.000,E1 251.040} C_DIS
LIN {X 0.277,Y -639.742,Z 316.190,A 0.000,B 0.000,C 90.000,E1 250.242} C_DIS
LIN {X 0.012,Y -639.571,Z 316.185,A 0.000,B 0.000,C 90.000,E1 249.263} C_DIS
LIN {X -0.073,Y -639.198,Z 316.181,A 0.000,B 0.000,C 90.000,E1 248.518} C_DIS
LIN {X 0.193,Y -638.450,Z 316.176,A 0.000,B 0.000,C 90.000,E1 247.741} C_DIS
LIN {X 0.093,Y -637.543,Z 316.172,A 0.000,B 0.000,C 90.000,E1 246.997} C_DIS
LIN {X 0.028,Y -635.861,Z 316.167,A 0.000,B 0.000,C 90.000,E1 245.997} C_DIS
LIN {X 0.205,Y -633.758,Z 316.161,A 0.000,B 0.000,C 90.000,E1 244.973} C_DIS
LIN {X 0.087,Y -631.280,Z 316.155,A 0.000,B 0.000,C 90.000,E1 243.973} C_DIS
LIN {X 0.206,Y -628.362,Z 316.150,A 0.000,B 0.000,C 90.000,E1 242.948} C_DIS
LIN {X -0.286,Y -626.090,Z 316.146,A 0.000,B 0.000,C 90.000,E1 242.231} C_DIS
LIN {X 0.064,Y -621.425,Z 316.137,A 0.000,B 0.000,C 90.000,E1 240.667} C_DIS
LIN {X 0.088,Y -616.590,Z 316.129,A 0.000,B 0.000,C 90.000,E1 239.125} C_DIS
LIN {X -0.025,Y -610.920,Z 316.119,A 0.000,B 0.000,C 90.000,E1 237.327} C_DIS
LIN {X 0.179,Y -606.859,Z 316.111,A 0.000,B 0.000,C 90.000,E1 236.008} C_DIS
LIN {X -0.014,Y -601.054,Z 316.101,A 0.000,B 0.000,C 90.000,E1 234.196} C_DIS
LIN {X -0.110,Y -598.499,Z 316.097,A 0.000,B 0.000,C 90.000,E1 233.417} C_DIS
LIN {X -0.245,Y -593.909,Z 316.089,A 0.000,B 0.000,C 90.000,E1 232.110} C_DIS
LIN {X -0.054,Y -587.569,Z 316.079,A 0.000,B 0.000,C 90.000,E1 230.231} C_DIS
LIN {X 0.367,Y -583.095,Z 316.072,A 0.000,B 0.000,C 90.000,E1 228.852} C_DIS
LIN {X -0.118,Y -576.293,Z 316.060,A 0.000,B 0.000,C 90.000,E1 226.743} C_DIS
LIN {X -0.022,Y -572.803,Z 316.054,A 0.000,B 0.000,C 90.000,E1 225.648} C_DIS
LIN {X 0.102,Y -565.041,Z 316.040,A 0.000,B 0.000,C 90.000,E1 223.176} C_DIS
LIN {X -0.286,Y -560.794,Z 316.032,A 0.000,B 0.000,C 90.000,E1 221.838} C_DIS
LIN {X -0.255,Y -555.673,Z 316.023,A 0.000,B 0.000,C 90.000,E1 220.172} C_DIS
LIN {X 0.087,Y -550.495,Z 316.014,A 0.000,B 0.000,C 90.000,E1 218.463} C_DIS
LIN {X -0.075,Y -546.383,Z 316.006,A 0.000,B 0.000,C 90.000,E1 217.076} C_DIS
LIN {X -0.081,Y -538.192,Z 315.990,A 0.000,B 0.000,C 90.000,E1 214.246} C_DIS
LIN {X 0.238,Y -532.895,Z 315.979,A 0.000,B 0.000,C 90.000,E1 212.212} C_DIS
LIN {X -0.001,Y -528.463,Z 315.970,A 0.000,B 0.000,C 90.000,E1 210.512} C_DIS
LIN {X -0.098,Y -524.854,Z 315.962,A 0.000,B 0.000,C 90.000,E1 209.077} C_DIS
LIN {X -0.114,Y -520.622,Z 315.952,A 0.000,B 0.000,C 90.000,E1 207.334} C_DIS
LIN {X -0.084,Y -514.589,Z 315.937,A 0.000,B 0.000,C 90.000,E1 204.695} C_DIS
LIN {X -0.190,Y -509.964,Z 315.926,A 0.000,B 0.000,C 90.000,E1 202.642} C_DIS
LIN {X -0.136,Y -506.706,Z 315.917,A 0.000,B 0.000,C 90.000,E1 201.153} C_DIS
LIN {X 0.228,Y -502.943,Z 315.908,A 0.000,B 0.000,C 90.000,E1 199.322} C_DIS
LIN {X 0.214,Y -497.448,Z 315.893,A 0.000,B 0.000,C 90.000,E1 196.622} C_DIS
LIN {X 0.026,Y -494.611,Z 315.884,A 0.000,B 0.000,C 90.000,E1 195.134} C_DIS
LIN {X -0.049,Y -490.506,Z 315.871,A 0.000,B 0.000,C 90.000,E1 192.715} C_DIS
LIN {X -0.126,Y -487.465,Z 315.861,A 0.000,B 0.000,C 90.000,E1 190.894} C_DIS
LIN {X 0.111,Y -483.206,Z 315.845,A 0.000,B 0.000,C 90.000,E1 188.106} C_DIS
LIN {X 0.065,Y -479.388,Z 315.830,A 0.000,B 0.000,C 90.000,E1 185.334} C_DIS
LIN {X 0.237,Y -476.038,Z 315.814,A 0.000,B 0.000,C 90.000,E1 182.522} C_DIS
LIN {X -0.127,Y -472.238,Z 315.792,A 0.000,B 0.000,C 90.000,E1 178.511} C_DIS
LIN {X -0.226,Y -470.822,Z 315.780,A 0.000,B 0.000,C 90.000,E1 176.331} C_DIS
LIN {X -0.048,Y -469.889,Z 315.766,A 0.000,B 0.000,C 90.000,E1 173.799} C_DIS
LIN {X -0.223,Y -469.373,Z 315.748,A 0.000,B 0.000,C 90.000,E1 170.679} C_DIS
LIN {X -0.016,Y -469.650,Z 315.732,A 0.000,B 0.000,C 90.000,E1 167.825} C_DIS
LIN {X -0.194,Y -470.876,Z 315.713,A 0.000,B 0.000,C 90.000,E1 164.393} C_DIS
LIN {X 0.000,Y -471.919,Z 315.703,A 0.000,B 0.000,C 90.000,E1 162.489} C_DIS
LIN {X -0.175,Y -473.739,Z 315.689,A 0.000,B 0.000,C 90.000,E1 160.007} C_DIS
LIN {X 0.120,Y -478.041,Z 315.666,A 0.000,B 0.000,C 90.000,E1 155.921} C_DIS
LIN {X -0.055,Y -483.065,Z 315.647,A 0.000,B 0.000,C 90.000,E1 152.538} C_DIS
LIN {X 0.006,Y -488.666,Z 315.630,A 0.000,B 0.000,C 90.000,E1 149.459} C_DIS
LIN {X 0.091,Y -494.667,Z 315.615,A 0.000,B 0.000,C 90.000,E1 146.707} C_DIS
LIN {X 0.216,Y -500.302,Z 315.602,A 0.000,B 0.000,C 90.000,E1 144.276} C_DIS
LIN {X 0.014,Y -503.598,Z 315.593,A 0.000,B 0.000,C 90.000,E1 142.798} C_DIS
LIN {X -0.120,Y -506.119,Z 315.587,A 0.000,B 0.000,C 90.000,E1 141.618} C_DIS
LIN {X -0.113,Y -507.834,Z 315.582,A 0.000,B 0.000,C 90.000,E1 140.723} C_DIS
LIN {X -0.181,Y -509.926,Z 315.575,A 0.000,B 0.000,C 90.000,E1 139.542} C_DIS
LIN {X 0.204,Y -511.365,Z 315.570,A 0.000,B 0.000,C 90.000,E1 138.609} C_DIS
LIN {X -0.204,Y -512.782,Z 315.564,A 0.000,B 0.000,C 90.000,E1 137.472} C_DIS
LIN {X -0.043,Y -513.371,Z 315.560,A 0.000,B 0.000,C 90.000,E1 136.863} C_DIS
LIN {X 0.011,Y -514.023,Z 315.555,A 0.000,B 0.000,C 90.000,E1 135.972} C_DIS
LIN {X 0.075,Y -514.287,Z 315.551,A 0.000,B 0.000,C 90.000,E1 135.081} C_DIS
LIN {X 0.143,Y -514.307,Z 315.546,A 0.000,B 0.000,C 90.000,E1 134.190} C_DIS
LIN {X -0.055,Y -514.231,Z 315.542,A 0.000,B 0.000,C 90.000,E1 133.623} C_DIS
LIN {X 0.004,Y -513.832,Z 315.537,A 0.000,B 0.000,C 90.000,E1 132.732} C_DIS
LIN {X 0.089,Y -513.168,Z 315.533,A 0.000,B 0.000,C 90.000,E1 131.838} C_DIS
LIN {X -0.211,Y -512.268,Z 315.528,A 0.000,B 0.000,C 90.000,E1 130.987} C_DIS
LIN {X -0.221,Y -510.744,Z 315.521,A 0.000,B 0.000,C 90.000,E1 129.806} C_DIS
LIN {X -0.021,Y -508.741,Z 315.513,A 0.000,B 0.000,C 90.000,E1 128.302} C_DIS
LIN {X 0.218,Y -506.638,Z 315.505,A 0.000,B 0.000,C 90.000,E1 126.790} C_DIS
LIN {X 0.222,Y -504.818,Z 315.498,A 0.000,B 0.000,C 90.000,E1 125.598} C_DIS
LIN {X 0.202,Y -502.703,Z 315.491,A 0.000,B 0.000,C 90.000,E1 124.405} C_DIS
LIN {X -0.130,Y -500.461,Z 315.485,A 0.000,B 0.000,C 90.000,E1 123.245} C_DIS
LIN {X 0.059,Y -497.524,Z 315.476,A 0.000,B 0.000,C 90.000,E1 121.720} C_DIS
LIN {X 0.089,Y -494.454,Z 315.468,A 0.000,B 0.000,C 90.000,E1 120.207} C_DIS
LIN {X 0.160,Y -489.472,Z 315.454,A 0.000,B 0.000,C 90.000,E1 117.769} C_DIS
LIN {X 0.245,Y -486.379,Z 315.446,A 0.000,B 0.000,C 90.000,E1 116.232} C_DIS
LIN {X -0.168,Y -482.013,Z 315.434,A 0.000,B 0.000,C 90.000,E1 114.131} C_DIS
LIN {X -0.190,Y -478.149,Z 315.424,A 0.000,B 0.000,C 90.000,E1 112.280} C_DIS
LIN {X 0.156,Y -474.394,Z 315.413,A 0.000,B 0.000,C 90.000,E1 110.375} C_DIS
LIN {X 0.033,Y -471.902,Z 315.406,A 0.000,B 0.000,C 90.000,E1 109.141} C_DIS
LIN {X -0.151,Y -467.558,Z 315.394,A 0.000,B 0.000,C 90.000,E1 106.968} C_DIS
LIN {X 0.106,Y -465.421,Z 315.388,A 0.000,B 0.000,C 90.000,E1 105.843} C_DIS
LIN {X 0.067,Y -465.433,Z 315.388,A 0.000,B 0.000,C 90.000,E1 105.843} C_DIS
LIN {X -0.063,Y -467.381,Z 315.384,A 0.000,B 0.000,C 90.000,E1 105.064} C_DIS
LIN {X 0.193,Y -468.024,Z 315.382,A 0.000,B 0.000,C 90.000,E1 104.717} C_DIS
LIN {X 0.170,Y -476.236,Z 315.356,A 0.000,B 0.000,C 90.000,E1 100.018} C_DIS
LIN {X -0.044,Y -482.131,Z 315.330,A 0.000,B 0.000,C 90.000,E1 95.391} C_DIS
LIN {X 0.191,Y -485.529,Z 315.304,A 0.000,B 0.000,C 90.000,E1 90.745} C_DIS
LIN {X 0.223,Y -486.380,Z 315.280,A 0.000,B 0.000,C 90.000,E1 86.445} C_DIS
LIN {X 0.048,Y -486.350,Z 315.279,A 0.000,B 0.000,C 90.000,E1 86.159} C_DIS
LIN {X 0.126,Y -484.665,Z 315.253,A 0.000,B 0.000,C 90.000,E1 81.546} C_DIS
LIN {X 0.016,Y -480.584,Z 315.227,A 0.000,B 0.000,C 90.000,E1 76.937} C_DIS
LIN {X -0.271,Y -479.659,Z 315.224,A 0.000,B 0.000,C 90.000,E1 76.353} C_DIS
LIN {X -0.241,Y -476.396,Z 315.212,A 0.000,B 0.000,C 90.000,E1 74.102} C_DIS
LIN {X -0.282,Y -476.391,Z 315.212,A 0.000,B 0.000,C 90.000,E1 74.102} C_DIS
LIN {X -0.167,Y -480.797,Z 315.202,A 0.000,B 0.000,C 90.000,E1 72.308} C_DIS
LIN {X 0.126,Y -486.380,Z 315.190,A 0.000,B 0.000,C 90.000,E1 70.115} C_DIS
LIN {X 0.030,Y -489.707,Z 315.183,A 0.000,B 0.000,C 90.000,E1 68.901} C_DIS
LIN {X 0.157,Y -493.090,Z 315.176,A 0.000,B 0.000,C 90.000,E1 67.667} C_DIS
LIN {X -0.020,Y -498.187,Z 315.166,A 0.000,B 0.000,C 90.000,E1 65.869} C_DIS
LIN {X -0.051,Y -504.221,Z 315.154,A 0.000,B 0.000,C 90.000,E1 63.768} C_DIS
LIN {X -0.101,Y -508.519,Z 315.146,A 0.000,B 0.000,C 90.000,E1 62.281} C_DIS
LIN {X 0.271,Y -513.696,Z 315.136,A 0.000,B 0.000,C 90.000,E1 60.461} C_DIS
LIN {X 0.198,Y -518.006,Z 315.128,A 0.000,B 0.000,C 90.000,E1 58.997} C_DIS
LIN {X -0.240,Y -522.253,Z 315.120,A 0.000,B 0.000,C 90.000,E1 57.582} C_DIS
LIN {X 0.080,Y -527.289,Z 315.110,A 0.000,B 0.000,C 90.000,E1 55.801} C_DIS
LIN {X 0.083,Y -531.244,Z 315.102,A 0.000,B 0.000,C 90.000,E1 54.356} C_DIS
LIN {X 0.043,Y -533.544,Z 315.097,A 0.000,B 0.000,C 90.000,E1 53.497} C_DIS
LIN {X 0.031,Y -536.388,Z 315.091,A 0.000,B 0.000,C 90.000,E1 52.351} C_DIS
LIN {X -0.030,Y -538.947,Z 315.085,A 0.000,B 0.000,C 90.000,E1 51.215} C_DIS
LIN {X 0.029,Y -541.312,Z 315.078,A 0.000,B 0.000,C 90.000,E1 50.070} C_DIS
LIN {X 0.044,Y -544.388,Z 315.069,A 0.000,B 0.000,C 90.000,E1 48.366} C_DIS
LIN {X -0.286,Y -545.732,Z 315.064,A 0.000,B 0.000,C 90.000,E1 47.553} C_DIS
LIN {X 0.161,Y -547.296,Z 315.058,A 0.000,B 0.000,C 90.000,E1 46.377} C_DIS
LIN {X -0.172,Y -548.299,Z 315.053,A 0.000,B 0.000,C 90.000,E1 45.567} C_DIS
LIN {X 0.284,Y -549.083,Z 315.048,A 0.000,B 0.000,C 90.000,E1 44.676} C_DIS
LIN {X 0.022,Y -550.037,Z 315.041,A 0.000,B 0.000,C 90.000,E1 43.299} C_DIS
LIN {X 0.160,Y -550.606,Z 315.034,A 0.000,B 0.000,C 90.000,E1 42.162} C_DIS
LIN {X -0.099,Y -550.887,Z 315.028,A 0.000,B 0.000,C 90.000,E1 41.067} C_DIS
LIN {X -0.001,Y -550.913,Z 315.023,A 0.000,B 0.000,C 90.000,E1 40.216} C_DIS
LIN {X -0.204,Y -550.571,Z 315.017,A 0.000,B 0.000,C 90.000,E1 39.116} C_DIS
LIN {X -0.033,Y -550.155,Z 315.013,A 0.000,B 0.000,C 90.000,E1 38.257} C_DIS
LIN {X -0.187,Y -549.162,Z 315.005,A 0.000,B 0.000,C 90.000,E1 36.870} C_DIS
LIN {X -0.029,Y -548.423,Z 315.000,A 0.000,B 0.000,C 90.000,E1 36.011} C_DIS
LIN {X -0.104,Y -547.104,Z 314.992,A 0.000,B 0.000,C 90.000,E1 34.612} C_DIS
LIN {X 0.285,Y -545.444,Z 314.983,A 0.000,B 0.000,C 90.000,E1 32.880} C_DIS
LIN {X 0.070,Y -543.553,Z 314.972,A 0.000,B 0.000,C 90.000,E1 30.924} C_DIS
LIN {X 0.263,Y -542.014,Z 314.962,A 0.000,B 0.000,C 90.000,E1 29.205} C_DIS
LIN {X -0.308,Y -540.780,Z 314.955,A 0.000,B 0.000,C 90.000,E1 27.847} C_DIS
LIN {X -0.225,Y -538.903,Z 314.944,A 0.000,B 0.000,C 90.000,E1 25.848} C_DIS
LIN {X -0.162,Y -537.324,Z 314.934,A 0.000,B 0.000,C 90.000,E1 24.131} C_DIS
LIN {X 0.131,Y -535.869,Z 314.924,A 0.000,B 0.000,C 90.000,E1 22.386} C_DIS
LIN {X -0.224,Y -535.067,Z 314.918,A 0.000,B 0.000,C 90.000,E1 21.280} C_DIS
LIN {X 0.038,Y -533.629,Z 314.905,A 0.000,B 0.000,C 90.000,E1 18.960} C_DIS
LIN {X -0.021,Y -532.934,Z 314.899,A 0.000,B 0.000,C 90.000,E1 17.819} C_DIS
LIN {X -0.165,Y -532.019,Z 314.886,A 0.000,B 0.000,C 90.000,E1 15.536} C_DIS
LIN {X 0.194,Y -531.415,Z 314.877,A 0.000,B 0.000,C 90.000,E1 13.772} C_DIS
LIN {X -0.004,Y -531.068,Z 314.869,A 0.000,B 0.000,C 90.000,E1 12.355} C_DIS
LIN {X -0.215,Y -530.925,Z 314.856,A 0.000,B 0.000,C 90.000,E1 10.074} C_DIS
LIN {X -0.056,Y -531.154,Z 314.841,A 0.000,B 0.000,C 90.000,E1 7.466} C_DIS
LIN {X -0.073,Y -531.854,Z 314.827,A 0.000,B 0.000,C 90.000,E1 4.878} C_DIS
LIN {X -0.075,Y -532.538,Z 314.819,A 0.000,B 0.000,C 90.000,E1 3.440} C_DIS
LIN {X -0.092,Y -533.606,Z 314.808,A 0.000,B 0.000,C 90.000,E1 1.432} C_DIS
LIN {X 0.202,Y -534.592,Z 314.799,A 0.000,B 0.000,C 90.000,E1 359.771} C_DIS
LIN {X 0.231,Y -537.000,Z 314.783,A 0.000,B 0.000,C 90.000,E1 356.906} C_DIS
LIN {X -0.223,Y -538.134,Z 314.777,A 0.000,B 0.000,C 90.000,E1 355.812} C_DIS
LIN {X 0.020,Y -540.832,Z 314.762,A 0.000,B 0.000,C 90.000,E1 353.223} C_DIS
LIN {X 0.127,Y -546.252,Z 314.745,A 0.000,B 0.000,C 90.000,E1 350.095} C_DIS
LIN {X -0.241,Y -550.970,Z 314.733,A 0.000,B 0.000,C 90.000,E1 347.881} C_DIS
LIN {X 0.169,Y -556.023,Z 314.722,A 0.000,B 0.000,C 90.000,E1 345.880} C_DIS
LIN {X -0.226,Y -561.363,Z 314.711,A 0.000,B 0.000,C 90.000,E1 343.976} C_DIS
LIN {X 0.214,Y -566.910,Z 314.700,A 0.000,B 0.000,C 90.000,E1 342.000} C_DIS
LIN {X -0.267,Y -570.944,Z 314.693,A 0.000,B 0.000,C 90.000,E1 340.678} C_DIS
LIN {X -0.123,Y -574.250,Z 314.686,A 0.000,B 0.000,C 90.000,E1 339.571} C_DIS
LIN {X 0.042,Y -582.959,Z 314.671,A 0.000,B 0.000,C 90.000,E1 336.847} C_DIS
LIN {X 0.107,Y -593.085,Z 314.655,A 0.000,B 0.000,C 90.000,E1 333.896} C_DIS
LIN {X -0.358,Y -597.838,Z 314.648,A 0.000,B 0.000,C 90.000,E1 332.615} C_DIS
LIN {X 0.135,Y -601.566,Z 314.642,A 0.000,B 0.000,C 90.000,E1 331.513} C_DIS
LIN {X 0.155,Y -605.217,Z 314.636,A 0.000,B 0.000,C 90.000,E1 330.461} C_DIS
LIN {X 0.224,Y -609.002,Z 314.630,A 0.000,B 0.000,C 90.000,E1 329.410} C_DIS
LIN {X -0.184,Y -612.697,Z 314.624,A 0.000,B 0.000,C 90.000,E1 328.408} C_DIS
LIN {X -0.257,Y -617.310,Z 314.617,A 0.000,B 0.000,C 90.000,E1 327.120} C_DIS
LIN {X 0.062,Y -622.529,Z 314.609,A 0.000,B 0.000,C 90.000,E1 325.548} C_DIS
LIN {X -0.014,Y -626.705,Z 314.602,A 0.000,B 0.000,C 90.000,E1 324.276} C_DIS
LIN {X 0.000,Y -629.823,Z 314.596,A 0.000,B 0.000,C 90.000,E1 323.256} C_DIS
LIN {X 0.048,Y -633.476,Z 314.589,A 0.000,B 0.000,C 90.000,E1 321.984} C_DIS
LIN {X -0.065,Y -637.792,Z 314.580,A 0.000,B 0.000,C 90.000,E1 320.481} C_DIS
LIN {X -0.080,Y -642.206,Z 314.572,A 0.000,B 0.000,C 90.000,E1 318.976} C_DIS
LIN {X 0.132,Y -645.095,Z 314.567,A 0.000,B 0.000,C 90.000,E1 317.957} C_DIS
LIN {X -0.063,Y -653.311,Z 314.551,A 0.000,B 0.000,C 90.000,E1 315.243} C_DIS
LIN {X -0.228,Y -656.215,Z 314.546,A 0.000,B 0.000,C 90.000,E1 314.271} C_DIS
LIN {X 0.094,Y -659.647,Z 314.539,A 0.000,B 0.000,C 90.000,E1 313.014} C_DIS
LIN {X 0.000,Y -662.247,Z 314.534,A 0.000,B 0.000,C 90.000,E1 312.043} C_DIS
LIN {X -0.016,Y -664.696,Z 314.528,A 0.000,B 0.000,C 90.000,E1 311.067} C_DIS
LIN {X 0.015,Y -666.459,Z 314.524,A 0.000,B 0.000,C 90.000,E1 310.334} C_DIS
LIN {X 0.055,Y -669.126,Z 314.517,A 0.000,B 0.000,C 90.000,E1 309.116} C_DIS
LIN {X 0.233,Y -671.544,Z 314.511,A 0.000,B 0.000,C 90.000,E1 307.890} C_DIS
LIN {X -0.191,Y -672.468,Z 314.508,A 0.000,B 0.000,C 90.000,E1 307.443} C_DIS
LIN {X 0.047,Y -673.968,Z 314.503,A 0.000,B 0.000,C 90.000,E1 306.457} C_DIS
LIN {X 0.167,Y -674.898,Z 314.499,A 0.000,B 0.000,C 90.000,E1 305.724} C_DIS
LIN {X -0.103,Y -675.621,Z 314.495,A 0.000,B 0.000,C 90.000,E1 305.025} C_DIS
LIN {X 0.193,Y -676.108,Z 314.491,A 0.000,B 0.000,C 90.000,E1 304.278} C_DIS
LIN {X 0.335,Y -676.311,Z 314.488,A 0.000,B 0.000,C 90.000,E1 303.785} C_DIS
LIN {X 0.246,Y -676.304,Z 314.483,A 0.000,B 0.000,C 90.000,E1 302.832} C_DIS
LIN {X -0.017,Y -676.123,Z 314.479,A 0.000,B 0.000,C 90.000,E1 302.133} C_DIS
LIN {X -0.067,Y -675.570,Z 314.475,A 0.000,B 0.000,C 90.000,E1 301.416} C_DIS
LIN {X 0.233,Y -674.706,Z 314.471,A 0.000,B 0.000,C 90.000,E1 300.669} C_DIS
LIN {X 0.180,Y -673.577,Z 314.467,A 0.000,B 0.000,C 90.000,E1 299.951} C_DIS
LIN {X -0.137,Y -672.215,Z 314.463,A 0.000,B 0.000,C 90.000,E1 299.255} C_DIS
LIN {X 0.115,Y -669.556,Z 314.456,A 0.000,B 0.000,C 90.000,E1 298.025} C_DIS
LIN {X 0.023,Y -666.643,Z 314.449,A 0.000,B 0.000,C 90.000,E1 296.821} C_DIS
LIN {X 0.040,Y -664.152,Z 314.444,A 0.000,B 0.000,C 90.000,E1 295.848} C_DIS
LIN {X -0.133,Y -660.916,Z 314.437,A 0.000,B 0.000,C 90.000,E1 294.643} C_DIS
LIN {X 0.241,Y -657.590,Z 314.430,A 0.000,B 0.000,C 90.000,E1 293.387} C_DIS
LIN {X -0.202,Y -653.506,Z 314.422,A 0.000,B 0.000,C 90.000,E1 291.950} C_DIS
LIN {X 0.248,Y -649.552,Z 314.414,A 0.000,B 0.000,C 90.000,E1 290.429} C_DIS
LIN {X -0.237,Y -643.887,Z 314.401,A 0.000,B 0.000,C 90.000,E1 288.236} C_DIS
LIN {X -0.046,Y -638.129,Z 314.387,A 0.000,B 0.000,C 90.000,E1 285.717} C_DIS
LIN {X 0.226,Y -633.162,Z 314.373,A 0.000,B 0.000,C 90.000,E1 283.175} C_DIS
LIN {X -0.037,Y -628.095,Z 314.355,A 0.000,B 0.000,C 90.000,E1 279.905} C_DIS
LIN {X 0.257,Y -625.460,Z 314.342,A 0.000,B 0.000,C 90.000,E1 277.587} C_DIS
LIN {X 0.242,Y -622.849,Z 314.322,A 0.000,B 0.000,C 90.000,E1 274.012} C_DIS
LIN {X 0.133,Y -622.072,Z 314.310,A 0.000,B 0.000,C 90.000,E1 271.718} C_DIS
LIN {X 0.273,Y -621.883,Z 314.298,A 0.000,B 0.000,C 90.000,E1 269.656} C_DIS
LIN {X 0.135,Y -622.375,Z 314.285,A 0.000,B 0.000,C 90.000,E1 267.364} C_DIS
LIN {X 0.085,Y -623.576,Z 314.273,A 0.000,B 0.000,C 90.000,E1 265.065} C_DIS
LIN {X 0.133,Y -625.351,Z 314.260,A 0.000,B 0.000,C 90.000,E1 262.761} C_DIS
LIN {X 0.196,Y -627.123,Z 314.250,A 0.000,B 0.000,C 90.000,E1 260.971} C_DIS
LIN {X -0.115,Y -629.212,Z 314.240,A 0.000,B 0.000,C 90.000,E1 259.218} C_DIS
LIN {X 0.063,Y -631.987,Z 314.229,A 0.000,B 0.000,C 90.000,E1 257.173} C_DIS
LIN {X -0.246,Y -633.839,Z 314.222,A 0.000,B 0.000,C 90.000,E1 255.936} C_DIS
LIN {X 0.248,Y -635.576,Z 314.215,A 0.000,B 0.000,C 90.000,E1 254.629} C_DIS
LIN {X -0.280,Y -636.386,Z 314.211,A 0.000,B 0.000,C 90.000,E1 253.921} C_DIS
LIN {X 0.261,Y -637.717,Z 314.202,A 0.000,B 0.000,C 90.000,E1 252.362} C_DIS
LIN {X -0.242,Y -638.403,Z 314.197,A 0.000,B 0.000,C 90.000,E1 251.402} C_DIS
LIN {X 0.250,Y -638.711,Z 314.192,A 0.000,B 0.000,C 90.000,E1 250.604} C_DIS
LIN {X -0.068,Y -638.751,Z 314.188,A 0.000,B 0.000,C 90.000,E1 249.880} C_DIS
LIN {X -0.349,Y -638.486,Z 314.183,A 0.000,B 0.000,C 90.000,E1 248.901} C_DIS
LIN {X 0.290,Y -638.405,Z 314.181,A 0.000,B 0.000,C 90.000,E1 248.592} C_DIS
LIN {X 0.000,Y -637.497,Z 314.176,A 0.000,B 0.000,C 90.000,E1 247.614} C_DIS
LIN {X 0.094,Y -636.928,Z 314.173,A 0.000,B 0.000,C 90.000,E1 247.102} C_DIS
LIN {X -0.017,Y -635.774,Z 314.169,A 0.000,B 0.000,C 90.000,E1 246.357} C_DIS
LIN {X -0.099,Y -633.958,Z 314.163,A 0.000,B 0.000,C 90.000,E1 245.357} C_DIS
LIN {X 0.061,Y -631.656,Z 314.157,A 0.000,B 0.000,C 90.000,E1 244.332} C_DIS
LIN {X -0.145,Y -630.407,Z 314.155,A 0.000,B 0.000,C 90.000,E1 243.845} C_DIS
LIN {X -0.018,Y -626.787,Z 314.148,A 0.000,B 0.000,C 90.000,E1 242.564} C_DIS
LIN {X -0.203,Y -621.386,Z 314.138,A 0.000,B 0.000,C 90.000,E1 240.795} C_DIS
LIN {X -0.197,Y -615.770,Z 314.128,A 0.000,B 0.000,C 90.000,E1 238.997} C_DIS
LIN {X -0.001,Y -610.091,Z 314.118,A 0.000,B 0.000,C 90.000,E1 237.168} C_DIS
LIN {X -0.142,Y -606.010,Z 314.110,A 0.000,B 0.000,C 90.000,E1 235.881} C_DIS
LIN {X -0.006,Y -600.238,Z 314.100,A 0.000,B 0.000,C 90.000,E1 234.036} C_DIS
LIN {X 0.133,Y -596.717,Z 314.094,A 0.000,B 0.000,C 90.000,E1 232.970} C_DIS
LIN {X 0.029,Y -590.292,Z 314.084,A 0.000,B 0.000,C 90.000,E1 231.126} C_DIS
LIN {X 0.114,Y -585.814,Z 314.077,A 0.000,B 0.000,C 90.000,E1 229.784} C_DIS
LIN {X -0.037,Y -579.688,Z 314.066,A 0.000,B 0.000,C 90.000,E1 227.919} C_DIS
LIN {X 0.248,Y -575.509,Z 314.059,A 0.000,B 0.000,C 90.000,E1 226.539} C_DIS
LIN {X -0.085,Y -571.981,Z 314.053,A 0.000,B 0.000,C 90.000,E1 225.486} C_DIS
LIN {X -0.084,Y -565.136,Z 314.041,A 0.000,B 0.000,C 90.000,E1 223.299} C_DIS
LIN {X -0.058,Y -560.930,Z 314.033,A 0.000,B 0.000,C 90.000,E1 221.919} C_DIS
LIN {X -0.025,Y -555.833,Z 314.024,A 0.000,B 0.000,C 90.000,E1 220.253} C_DIS
LIN {X -0.110,Y -550.691,Z 314.014,A 0.000,B 0.000,C 90.000,E1 218.588} C_DIS
LIN {X 0.163,Y -546.548,Z 314.007,A 0.000,B 0.000,C 90.000,E1 217.156} C_DIS
LIN {X 0.165,Y -538.330,Z 313.991,A 0.000,B 0.000,C 90.000,E1 214.326} C_DIS
LIN {X 0.051,Y -534.473,Z 313.983,A 0.000,B 0.000,C 90.000,E1 212.911} C_DIS
LIN {X -0.139,Y -529.962,Z 313.973,A 0.000,B 0.000,C 90.000,E1 211.209} C_DIS
LIN {X 0.013,Y -525.621,Z 313.964,A 0.000,B 0.000,C 90.000,E1 209.461} C_DIS
LIN {X -0.072,Y -520.621,Z 313.952,A 0.000,B 0.000,C 90.000,E1 207.436} C_DIS
LIN {X 0.188,Y -514.547,Z 313.938,A 0.000,B 0.000,C 90.000,E1 204.771} C_DIS
LIN {X 0.087,Y -509.927,Z 313.926,A 0.000,B 0.000,C 90.000,E1 202.717} C_DIS
LIN {X 0.244,Y -506.033,Z 313.916,A 0.000,B 0.000,C 90.000,E1 200.918} C_DIS
LIN {X 0.122,Y -502.297,Z 313.906,A 0.000,B 0.000,C 90.000,E1 199.141} C_DIS
LIN {X 0.183,Y -497.517,Z 313.893,A 0.000,B 0.000,C 90.000,E1 196.732} C_DIS
LIN {X -0.108,Y -494.137,Z 313.883,A 0.000,B 0.000,C 90.000,E1 194.954} C_DIS
LIN {X -0.093,Y -490.671,Z 313.871,A 0.000,B 0.000,C 90.000,E1 192.827} C_DIS
LIN {X -0.172,Y -487.676,Z 313.861,A 0.000,B 0.000,C 90.000,E1 191.007} C_DIS
LIN {X 0.067,Y -483.528,Z 313.846,A 0.000,B 0.000,C 90.000,E1 188.219} C_DIS
LIN {X -0.018,Y -479.803,Z 313.830,A 0.000,B 0.000,C 90.000,E1 185.454} C_DIS
LIN {X 0.210,Y -476.473,Z 313.815,A 0.000,B 0.000,C 90.000,E1 182.636} C_DIS
LIN {X -0.123,Y -475.130,Z 313.808,A 0.000,B 0.000,C 90.000,E1 181.432} C_DIS
LIN {X 0.175,Y -472.151,Z 313.787,A 0.000,B 0.000,C 90.000,E1 177.650} C_DIS
LIN {X -0.016,Y -470.447,Z 313.766,A 0.000,B 0.000,C 90.000,E1 173.913} C_DIS
LIN {X 0.167,Y -470.009,Z 313.756,A 0.000,B 0.000,C 90.000,E1 172.008} C_DIS
LIN {X -0.135,Y -469.954,Z 313.740,A 0.000,B 0.000,C 90.000,E1 169.218} C_DIS
LIN {X -0.083,Y -470.357,Z 313.726,A 0.000,B 0.000,C 90.000,E1 166.700} C_DIS
LIN {X 0.197,Y -471.429,Z 313.712,A 0.000,B 0.000,C 90.000,E1 164.157} C_DIS
LIN {X -0.091,Y -472.729,Z 313.700,A 0.000,B 0.000,C 90.000,E1 162.000} C_DIS
LIN {X -0.268,Y -474.803,Z 313.684,A 0.000,B 0.000,C 90.000,E1 159.209} C_DIS
LIN {X 0.164,Y -477.376,Z 313.671,A 0.000,B 0.000,C 90.000,E1 156.666} C_DIS
LIN {X -0.009,Y -481.064,Z 313.655,A 0.000,B 0.000,C 90.000,E1 153.896} C_DIS
LIN {X 0.157,Y -486.087,Z 313.638,A 0.000,B 0.000,C 90.000,E1 150.795} C_DIS
LIN {X -0.018,Y -492.870,Z 313.619,A 0.000,B 0.000,C 90.000,E1 147.454} C_DIS
LIN {X 0.058,Y -496.174,Z 313.611,A 0.000,B 0.000,C 90.000,E1 145.928} C_DIS
LIN {X 0.073,Y -500.368,Z 313.601,A 0.000,B 0.000,C 90.000,E1 144.116} C_DIS
LIN {X -0.123,Y -503.566,Z 313.592,A 0.000,B 0.000,C 90.000,E1 142.637} C_DIS
LIN {X 0.141,Y -506.033,Z 313.586,A 0.000,B 0.000,C 90.000,E1 141.412} C_DIS
LIN {X 0.044,Y -508.202,Z 313.579,A 0.000,B 0.000,C 90.000,E1 140.231} C_DIS
LIN {X -0.078,Y -510.164,Z 313.573,A 0.000,B 0.000,C 90.000,E1 139.057} C_DIS
LIN {X 0.070,Y -510.994,Z 313.569,A 0.000,B 0.000,C 90.000,E1 138.447} C_DIS
LIN {X 0.130,Y -512.034,Z 313.564,A 0.000,B 0.000,C 90.000,E1 137.553} C_DIS
LIN {X -0.089,Y -512.654,Z 313.561,A 0.000,B 0.000,C 90.000,E1 136.986} C_DIS
LIN {X 0.331,Y -513.308,Z 313.556,A 0.000,B 0.000,C 90.000,E1 136.053} C_DIS
LIN {X 0.025,Y -513.610,Z 313.551,A 0.000,B 0.000,C 90.000,E1 135.202} C_DIS
LIN {X -0.279,Y -513.610,Z 313.546,A 0.000,B 0.000,C 90.000,E1 134.352} C_DIS
LIN {X -0.221,Y -513.418,Z 313.541,A 0.000,B 0.000,C 90.000,E1 133.461} C_DIS
LIN {X 0.206,Y -512.981,Z 313.536,A 0.000,B 0.000,C 90.000,E1 132.528} C_DIS
LIN {X -0.095,Y -512.247,Z 313.532,A 0.000,B 0.000,C 90.000,E1 131.676} C_DIS
LIN {X -0.020,Y -511.289,Z 313.527,A 0.000,B 0.000,C 90.000,E1 130.782} C_DIS
LIN {X 0.286,Y -509.742,Z 313.520,A 0.000,B 0.000,C 90.000,E1 129.564} C_DIS
LIN {X 0.239,Y -508.154,Z 313.513,A 0.000,B 0.000,C 90.000,E1 128.382} C_DIS
LIN {X -0.241,Y -506.071,Z 313.505,A 0.000,B 0.000,C 90.000,E1 126.950} C_DIS
LIN {X 0.055,Y -504.244,Z 313.499,A 0.000,B 0.000,C 90.000,E1 125.724} C_DIS
LIN {X 0.137,Y -502.680,Z 313.494,A 0.000,B 0.000,C 90.000,E1 124.818} C_DIS
LIN {X 0.081,Y -500.463,Z 313.487,A 0.000,B 0.000,C 90.000,E1 123.627} C_DIS
LIN {X 0.281,Y -496.969,Z 313.477,A 0.000,B 0.000,C 90.000,E1 121.799} C_DIS
LIN {X 0.144,Y -493.289,Z 313.467,A 0.000,B 0.000,C 90.000,E1 120.001} C_DIS
LIN {X -0.054,Y -488.326,Z 313.453,A 0.000,B 0.000,C 90.000,E1 117.590} C_DIS
LIN {X 0.018,Y -485.250,Z 313.445,A 0.000,B 0.000,C 90.000,E1 116.052} C_DIS
LIN {X 0.024,Y -480.921,Z 313.433,A 0.000,B 0.000,C 90.000,E1 113.898} C_DIS
LIN {X 0.166,Y -477.088,Z 313.423,A 0.000,B 0.000,C 90.000,E1 112.025} C_DIS
LIN {X 0.063,Y -473.981,Z 313.414,A 0.000,B 0.000,C 90.000,E1 110.482} C_DIS
LIN {X -0.227,Y -471.543,Z 313.407,A 0.000,B 0.000,C 90.000,E1 109.268} C_DIS
LIN {X 0.035,Y -467.262,Z 313.395,A 0.000,B 0.000,C 90.000,E1 107.040} C_DIS
LIN {X -0.114,Y -465.198,Z 313.389,A 0.000,B 0.000,C 90.000,E1 105.969} C_DIS
LIN {X -0.026,Y -465.197,Z 313.389,A 0.000,B 0.000,C 90.000,E1 105.953} C_DIS
LIN {X 0.050,Y -467.891,Z 313.382,A 0.000,B 0.000,C 90.000,E1 104.828} C_DIS
LIN {X 0.079,Y -475.456,Z 313.358,A 0.000,B 0.000,C 90.000,E1 100.433} C_DIS
LIN {X -0.084,Y -476.104,Z 313.356,A 0.000,B 0.000,C 90.000,E1 100.141} C_DIS
LIN {X 0.200,Y -482.022,Z 313.330,A 0.000,B 0.000,C 90.000,E1 95.454} C_DIS
LIN {X 0.129,Y -483.061,Z 313.320,A 0.000,B 0.000,C 90.000,E1 93.612} C_DIS
LIN {X -0.009,Y -485.462,Z 313.305,A 0.000,B 0.000,C 90.000,E1 90.859} C_DIS
LIN {X -0.219,Y -485.510,Z 313.298,A 0.000,B 0.000,C 90.000,E1 89.656} C_DIS
LIN {X 0.023,Y -486.384,Z 313.281,A 0.000,B 0.000,C 90.000,E1 86.560} C_DIS
LIN {X -0.152,Y -486.364,Z 313.279,A 0.000,B 0.000,C 90.000,E1 86.274} C_DIS
LIN {X -0.064,Y -484.690,Z 313.254,A 0.000,B 0.000,C 90.000,E1 81.659} C_DIS
LIN {X 0.082,Y -484.059,Z 313.250,A 0.000,B 0.000,C 90.000,E1 81.027} C_DIS
LIN {X -0.153,Y -480.633,Z 313.228,A 0.000,B 0.000,C 90.000,E1 77.048} C_DIS
LIN {X 0.173,Y -480.325,Z 313.226,A 0.000,B 0.000,C 90.000,E1 76.700} C_DIS
LIN {X -0.111,Y -476.187,Z 313.211,A 0.000,B 0.000,C 90.000,E1 73.921} C_DIS
LIN {X -0.151,Y -476.190,Z 313.211,A 0.000,B 0.000,C 90.000,E1 73.921} C_DIS
LIN {X 0.136,Y -479.940,Z 313.202,A 0.000,B 0.000,C 90.000,E1 72.362} C_DIS
LIN {X -0.207,Y -485.426,Z 313.190,A 0.000,B 0.000,C 90.000,E1 70.242} C_DIS
LIN {X 0.133,Y -488.763,Z 313.183,A 0.000,B 0.000,C 90.000,E1 68.975} C_DIS
LIN {X -0.180,Y -492.960,Z 313.175,A 0.000,B 0.000,C 90.000,E1 67.486} C_DIS
LIN {X -0.161,Y -498.050,Z 313.165,A 0.000,B 0.000,C 90.000,E1 65.665} C_DIS
LIN {X -0.031,Y -503.214,Z 313.155,A 0.000,B 0.000,C 90.000,E1 63.845} C_DIS
LIN {X -0.105,Y -507.563,Z 313.146,A 0.000,B 0.000,C 90.000,E1 62.359} C_DIS
LIN {X -0.209,Y -512.702,Z 313.137,A 0.000,B 0.000,C 90.000,E1 60.589} C_DIS
LIN {X 0.142,Y -517.050,Z 313.128,A 0.000,B 0.000,C 90.000,E1 59.076} C_DIS
LIN {X 0.062,Y -522.170,Z 313.119,A 0.000,B 0.000,C 90.000,E1 57.327} C_DIS
LIN {X -0.062,Y -527.148,Z 313.109,A 0.000,B 0.000,C 90.000,E1 55.595} C_DIS
LIN {X 0.247,Y -531.109,Z 313.101,A 0.000,B 0.000,C 90.000,E1 54.116} C_DIS
LIN {X -0.114,Y -534.125,Z 313.094,A 0.000,B 0.000,C 90.000,E1 53.004} C_DIS
LIN {X 0.208,Y -536.840,Z 313.088,A 0.000,B 0.000,C 90.000,E1 51.823} C_DIS
LIN {X -0.179,Y -539.321,Z 313.082,A 0.000,B 0.000,C 90.000,E1 50.723} C_DIS
LIN {X -0.154,Y -540.470,Z 313.079,A 0.000,B 0.000,C 90.000,E1 50.150} C_DIS
LIN {X 0.245,Y -543.570,Z 313.069,A 0.000,B 0.000,C 90.000,E1 48.405} C_DIS
LIN {X 0.270,Y -544.934,Z 313.064,A 0.000,B 0.000,C 90.000,E1 47.553} C_DIS
LIN {X -0.067,Y -546.522,Z 313.058,A 0.000,B 0.000,C 90.000,E1 46.458} C_DIS
LIN {X -0.016,Y -547.555,Z 313.053,A 0.000,B 0.000,C 90.000,E1 45.607} C_DIS
LIN {X 0.039,Y -548.372,Z 313.049,A 0.000,B 0.000,C 90.000,E1 44.757} C_DIS
LIN {X -0.200,Y -549.500,Z 313.039,A 0.000,B 0.000,C 90.000,E1 43.095} C_DIS
LIN {X 0.305,Y -550.029,Z 313.033,A 0.000,B 0.000,C 90.000,E1 41.919} C_DIS
LIN {X 0.033,Y -550.267,Z 313.027,A 0.000,B 0.000,C 90.000,E1 40.825} C_DIS
LIN {X 0.136,Y -550.320,Z 313.024,A 0.000,B 0.000,C 90.000,E1 40.253} C_DIS
LIN {X 0.280,Y -550.035,Z 313.018,A 0.000,B 0.000,C 90.000,E1 39.116} C_DIS
LIN {X 0.013,Y -549.651,Z 313.013,A 0.000,B 0.000,C 90.000,E1 38.302} C_DIS
LIN {X 0.229,Y -548.899,Z 313.007,A 0.000,B 0.000,C 90.000,E1 37.156} C_DIS
LIN {X -0.332,Y -547.984,Z 313.000,A 0.000,B 0.000,C 90.000,E1 36.091} C_DIS
LIN {X 0.083,Y -546.398,Z 312.991,A 0.000,B 0.000,C 90.000,E1 34.358} C_DIS
LIN {X 0.006,Y -544.762,Z 312.982,A 0.000,B 0.000,C 90.000,E1 32.673} C_DIS
LIN {X -0.022,Y -542.646,Z 312.969,A 0.000,B 0.000,C 90.000,E1 30.413} C_DIS
LIN {X -0.103,Y -540.846,Z 312.958,A 0.000,B 0.000,C 90.000,E1 28.437} C_DIS
LIN {X 0.304,Y -539.777,Z 312.952,A 0.000,B 0.000,C 90.000,E1 27.257} C_DIS
LIN {X -0.095,Y -538.184,Z 312.942,A 0.000,B 0.000,C 90.000,E1 25.591} C_DIS
LIN {X -0.055,Y -536.385,Z 312.931,A 0.000,B 0.000,C 90.000,E1 23.590} C_DIS
LIN {X 0.146,Y -534.589,Z 312.918,A 0.000,B 0.000,C 90.000,E1 21.280} C_DIS
LIN {X -0.112,Y -533.120,Z 312.906,A 0.000,B 0.000,C 90.000,E1 19.014} C_DIS
LIN {X 0.252,Y -531.878,Z 312.893,A 0.000,B 0.000,C 90.000,E1 16.677} C_DIS
LIN {X 0.199,Y -531.337,Z 312.885,A 0.000,B 0.000,C 90.000,E1 15.245} C_DIS
LIN {X -0.003,Y -530.860,Z 312.877,A 0.000,B 0.000,C 90.000,E1 13.828} C_DIS
LIN {X -0.215,Y -530.508,Z 312.869,A 0.000,B 0.000,C 90.000,E1 12.411} C_DIS
LIN {X 0.020,Y -530.314,Z 312.854,A 0.000,B 0.000,C 90.000,E1 9.792} C_DIS
LIN {X 0.177,Y -530.566,Z 312.840,A 0.000,B 0.000,C 90.000,E1 7.182} C_DIS
LIN {X 0.178,Y -531.210,Z 312.827,A 0.000,B 0.000,C 90.000,E1 4.878} C_DIS
LIN {X 0.150,Y -531.977,Z 312.818,A 0.000,B 0.000,C 90.000,E1 3.154} C_DIS
LIN {X 0.130,Y -532.920,Z 312.808,A 0.000,B 0.000,C 90.000,E1 1.432} C_DIS
LIN {X 0.199,Y -534.088,Z 312.797,A 0.000,B 0.000,C 90.000,E1 359.484} C_DIS
LIN {X 0.205,Y -536.003,Z 312.785,A 0.000,B 0.000,C 90.000,E1 357.192} C_DIS
LIN {X 0.278,Y -537.387,Z 312.777,A 0.000,B 0.000,C 90.000,E1 355.755} C_DIS
LIN {X -0.158,Y -539.063,Z 312.767,A 0.000,B 0.000,C 90.000,E1 354.090} C_DIS
LIN {X 0.023,Y -540.498,Z 312.761,A 0.000,B 0.000,C 90.000,E1 352.932} C_DIS
LIN {X -0.223,Y -543.816,Z 312.750,A 0.000,B 0.000,C 90.000,E1 350.971} C_DIS
LIN {X -0.253,Y -550.786,Z 312.731,A 0.000,B 0.000,C 90.000,E1 347.589} C_DIS
LIN {X 0.029,Y -555.136,Z 312.722,A 0.000,B 0.000,C 90.000,E1 345.880} C_DIS
LIN {X 0.148,Y -560.438,Z 312.711,A 0.000,B 0.000,C 90.000,E1 343.921} C_DIS
LIN {X 0.023,Y -565.959,Z 312.700,A 0.000,B 0.000,C 90.000,E1 342.000} C_DIS
LIN {X 0.251,Y -569.960,Z 312.692,A 0.000,B 0.000,C 90.000,E1 340.604} C_DIS
LIN {X -0.165,Y -572.471,Z 312.688,A 0.000,B 0.000,C 90.000,E1 339.826} C_DIS
LIN {X 0.013,Y -573.971,Z 312.685,A 0.000,B 0.000,C 90.000,E1 339.263} C_DIS
LIN {X -0.164,Y -576.647,Z 312.680,A 0.000,B 0.000,C 90.000,E1 338.465} C_DIS
LIN {X 0.314,Y -581.986,Z 312.671,A 0.000,B 0.000,C 90.000,E1 336.794} C_DIS
LIN {X -0.048,Y -586.436,Z 312.664,A 0.000,B 0.000,C 90.000,E1 335.485} C_DIS
LIN {X -0.301,Y -593.111,Z 312.653,A 0.000,B 0.000,C 90.000,E1 333.640} C_DIS
LIN {X -0.044,Y -598.778,Z 312.645,A 0.000,B 0.000,C 90.000,E1 332.025} C_DIS
LIN {X -0.130,Y -603.379,Z 312.637,A 0.000,B 0.000,C 90.000,E1 330.717} C_DIS
LIN {X -0.025,Y -606.109,Z 312.633,A 0.000,B 0.000,C 90.000,E1 329.921} C_DIS
LIN {X 0.110,Y -608.968,Z 312.629,A 0.000,B 0.000,C 90.000,E1 329.125} C_DIS
LIN {X -0.058,Y -614.459,Z 312.620,A 0.000,B 0.000,C 90.000,E1 327.582} C_DIS
LIN {X -0.062,Y -618.065,Z 312.614,A 0.000,B 0.000,C 90.000,E1 326.548} C_DIS
LIN {X 0.280,Y -623.308,Z 312.606,A 0.000,B 0.000,C 90.000,E1 324.975} C_DIS
LIN {X -0.096,Y -625.824,Z 312.601,A 0.000,B 0.000,C 90.000,E1 324.242} C_DIS
LIN {X 0.044,Y -628.988,Z 312.596,A 0.000,B 0.000,C 90.000,E1 323.210} C_DIS
LIN {X -0.040,Y -632.681,Z 312.589,A 0.000,B 0.000,C 90.000,E1 321.949} C_DIS
LIN {X -0.070,Y -637.012,Z 312.580,A 0.000,B 0.000,C 90.000,E1 320.436} C_DIS
LIN {X -0.111,Y -641.440,Z 312.572,A 0.000,B 0.000,C 90.000,E1 318.933} C_DIS
LIN {X 0.035,Y -644.316,Z 312.566,A 0.000,B 0.000,C 90.000,E1 317.919} C_DIS
LIN {X 0.296,Y -652.507,Z 312.551,A 0.000,B 0.000,C 90.000,E1 315.162} C_DIS
LIN {X 0.123,Y -655.403,Z 312.546,A 0.000,B 0.000,C 90.000,E1 314.190} C_DIS
LIN {X -0.050,Y -658.775,Z 312.539,A 0.000,B 0.000,C 90.000,E1 312.975} C_DIS
LIN {X -0.138,Y -661.998,Z 312.532,A 0.000,B 0.000,C 90.000,E1 311.757} C_DIS
LIN {X -0.152,Y -664.420,Z 312.527,A 0.000,B 0.000,C 90.000,E1 310.782} C_DIS
LIN {X -0.144,Y -667.174,Z 312.520,A 0.000,B 0.000,C 90.000,E1 309.564} C_DIS
LIN {X 0.001,Y -669.652,Z 312.513,A 0.000,B 0.000,C 90.000,E1 308.338} C_DIS
LIN {X 0.078,Y -671.450,Z 312.508,A 0.000,B 0.000,C 90.000,E1 307.363} C_DIS
LIN {X 0.301,Y -672.926,Z 312.502,A 0.000,B 0.000,C 90.000,E1 306.377} C_DIS
LIN {X 0.000,Y -674.115,Z 312.497,A 0.000,B 0.000,C 90.000,E1 305.438} C_DIS
LIN {X 0.277,Y -674.739,Z 312.493,A 0.000,B 0.000,C 90.000,E1 304.692} C_DIS
LIN {X 0.007,Y -675.119,Z 312.489,A 0.000,B 0.000,C 90.000,E1 303.992} C_DIS
LIN {X -0.132,Y -675.092,Z 312.482,A 0.000,B 0.000,C 90.000,E1 302.801} C_DIS
LIN {X -0.200,Y -674.886,Z 312.478,A 0.000,B 0.000,C 90.000,E1 302.084} C_DIS
LIN {X 0.094,Y -674.252,Z 312.474,A 0.000,B 0.000,C 90.000,E1 301.337} C_DIS
LIN {X 0.377,Y -673.340,Z 312.470,A 0.000,B 0.000,C 90.000,E1 300.590} C_DIS
LIN {X -0.105,Y -671.746,Z 312.465,A 0.000,B 0.000,C 90.000,E1 299.667} C_DIS
LIN {X -0.186,Y -670.222,Z 312.461,A 0.000,B 0.000,C 90.000,E1 298.949} C_DIS
LIN {X -0.117,Y -668.072,Z 312.455,A 0.000,B 0.000,C 90.000,E1 297.975} C_DIS
LIN {X 0.075,Y -665.135,Z 312.449,A 0.000,B 0.000,C 90.000,E1 296.744} C_DIS
LIN {X -0.079,Y -662.013,Z 312.442,A 0.000,B 0.000,C 90.000,E1 295.540} C_DIS
LIN {X -0.281,Y -658.723,Z 312.435,A 0.000,B 0.000,C 90.000,E1 294.335} C_DIS
LIN {X 0.169,Y -654.683,Z 312.427,A 0.000,B 0.000,C 90.000,E1 292.823} C_DIS
LIN {X 0.084,Y -651.964,Z 312.421,A 0.000,B 0.000,C 90.000,E1 291.844} C_DIS
LIN {X 0.056,Y -648.696,Z 312.415,A 0.000,B 0.000,C 90.000,E1 290.610} C_DIS
LIN {X 0.156,Y -643.002,Z 312.402,A 0.000,B 0.000,C 90.000,E1 288.362} C_DIS
LIN {X -0.016,Y -636.133,Z 312.385,A 0.000,B 0.000,C 90.000,E1 285.371} C_DIS
LIN {X 0.253,Y -630.014,Z 312.367,A 0.000,B 0.000,C 90.000,E1 282.063} C_DIS
LIN {X -0.245,Y -625.476,Z 312.349,A 0.000,B 0.000,C 90.000,E1 278.803} C_DIS
LIN {X 0.057,Y -622.415,Z 312.330,A 0.000,B 0.000,C 90.000,E1 275.454} C_DIS
LIN {X 0.049,Y -621.060,Z 312.315,A 0.000,B 0.000,C 90.000,E1 272.636} C_DIS
LIN {X 0.201,Y -620.666,Z 312.300,A 0.000,B 0.000,C 90.000,E1 270.057} C_DIS
LIN {X -0.246,Y -621.296,Z 312.283,A 0.000,B 0.000,C 90.000,E1 267.020} C_DIS
LIN {X -0.037,Y -622.433,Z 312.272,A 0.000,B 0.000,C 90.000,E1 264.951} C_DIS
LIN {X -0.029,Y -624.276,Z 312.259,A 0.000,B 0.000,C 90.000,E1 262.648} C_DIS
LIN {X -0.301,Y -625.803,Z 312.251,A 0.000,B 0.000,C 90.000,E1 261.141} C_DIS
LIN {X 0.077,Y -628.570,Z 312.238,A 0.000,B 0.000,C 90.000,E1 258.814} C_DIS
LIN {X -0.196,Y -631.088,Z 312.228,A 0.000,B 0.000,C 90.000,E1 257.061} C_DIS
LIN {X 0.242,Y -632.934,Z 312.221,A 0.000,B 0.000,C 90.000,E1 255.755} C_DIS
LIN {X 0.124,Y -634.376,Z 312.215,A 0.000,B 0.000,C 90.000,E1 254.755} C_DIS
LIN {X -0.242,Y -635.245,Z 312.211,A 0.000,B 0.000,C 90.000,E1 254.031} C_DIS
LIN {X 0.092,Y -636.584,Z 312.203,A 0.000,B 0.000,C 90.000,E1 252.489} C_DIS
LIN {X -0.225,Y -637.315,Z 312.197,A 0.000,B 0.000,C 90.000,E1 251.511} C_DIS
LIN {X 0.228,Y -637.617,Z 312.194,A 0.000,B 0.000,C 90.000,E1 250.967} C_DIS
LIN {X -0.281,Y -637.768,Z 312.189,A 0.000,B 0.000,C 90.000,E1 250.007} C_DIS
LIN {X 0.247,Y -637.606,Z 312.183,A 0.000,B 0.000,C 90.000,E1 248.954} C_DIS
LIN {X 0.101,Y -637.398,Z 312.180,A 0.000,B 0.000,C 90.000,E1 248.465} C_DIS
LIN {X -0.201,Y -636.508,Z 312.175,A 0.000,B 0.000,C 90.000,E1 247.486} C_DIS
LIN {X -0.318,Y -635.541,Z 312.171,A 0.000,B 0.000,C 90.000,E1 246.741} C_DIS
LIN {X -0.187,Y -634.332,Z 312.166,A 0.000,B 0.000,C 90.000,E1 245.973} C_DIS
LIN {X -0.326,Y -632.877,Z 312.162,A 0.000,B 0.000,C 90.000,E1 245.229} C_DIS
LIN {X -0.178,Y -630.547,Z 312.157,A 0.000,B 0.000,C 90.000,E1 244.204} C_DIS
LIN {X -0.114,Y -629.270,Z 312.154,A 0.000,B 0.000,C 90.000,E1 243.691} C_DIS
LIN {X 0.007,Y -625.679,Z 312.147,A 0.000,B 0.000,C 90.000,E1 242.410} C_DIS
